LIN {X 0.134,Y -371.526,Z 1771.538,A 0.000,B 0.000,C 90.000,E1 276.777} C_DIS
LIN {X 0.079,Y -367.433,Z 1771.535,A 0.000,B 0.000,C 90.000,E1 276.201} C_DIS
LIN {X 0.001,Y -362.698,Z 1771.531,A 0.000,B 0.000,C 90.000,E1 275.625} C_DIS
LIN {X -0.100,Y -357.339,Z 1771.528,A 0.000,B 0.000,C 90.000,E1 275.049} C_DIS
LIN {X -0.055,Y -351.569,Z 1771.525,A 0.000,B 0.000,C 90.000,E1 274.473} C_DIS
LIN {X -0.094,Y -345.659,Z 1771.522,A 0.000,B 0.000,C 90.000,E1 273.955} C_DIS
LIN {X 0.022,Y -339.520,Z 1771.519,A 0.000,B 0.000,C 90.000,E1 273.440} C_DIS
LIN {X 0.107,Y -330.116,Z 1771.515,A 0.000,B 0.000,C 90.000,E1 272.751} C_DIS
LIN {X 0.126,Y -323.725,Z 1771.513,A 0.000,B 0.000,C 90.000,E1 272.350} C_DIS
LIN {X 0.041,Y -317.098,Z 1771.511,A 0.000,B 0.000,C 90.000,E1 272.007} C_DIS
LIN {X -0.145,Y -310.058,Z 1771.509,A 0.000,B 0.000,C 90.000,E1 271.718} C_DIS
LIN {X -0.066,Y -302.742,Z 1771.508,A 0.000,B 0.000,C 90.000,E1 271.432} C_DIS
LIN {X -0.016,Y -295.334,Z 1771.507,A 0.000,B 0.000,C 90.000,E1 271.203} C_DIS
LIN {X 0.096,Y -283.998,Z 1771.505,A 0.000,B 0.000,C 90.000,E1 270.917} C_DIS
LIN {X -0.066,Y -272.910,Z 1771.504,A 0.000,B 0.000,C 90.000,E1 270.745} C_DIS
LIN {X -0.128,Y -259.523,Z 1771.503,A 0.000,B 0.000,C 90.000,E1 270.573} C_DIS
LIN {X 0.061,Y -245.252,Z 1771.502,A 0.000,B 0.000,C 90.000,E1 270.401} C_DIS
LIN {X 0.075,Y -232.395,Z 1771.502,A 0.000,B 0.000,C 90.000,E1 270.344} C_DIS
LIN {X 0.040,Y -181.579,Z 1771.502,A 0.000,B 0.000,C 90.000,E1 270.344} C_DIS
LIN {X 0.016,Y -180.851,Z 1771.472,A 0.000,B 0.000,C 90.000,E1 264.951} C_DIS
LIN {X 0.098,Y -178.961,Z 1771.444,A 0.000,B 0.000,C 90.000,E1 259.859} C_DIS
LIN {X -0.011,Y -177.369,Z 1771.430,A 0.000,B 0.000,C 90.000,E1 257.353} C_DIS
LIN {X 0.085,Y -175.543,Z 1771.411,A 0.000,B 0.000,C 90.000,E1 253.921} C_DIS
LIN {X -0.076,Y -172.276,Z 1771.387,A 0.000,B 0.000,C 90.000,E1 249.699} C_DIS
LIN {X -0.036,Y -171.755,Z 1771.382,A 0.000,B 0.000,C 90.000,E1 248.827} C_DIS
LIN {X -0.019,Y -167.355,Z 1771.354,A 0.000,B 0.000,C 90.000,E1 243.640} C_DIS
LIN {X 0.063,Y -166.743,Z 1771.349,A 0.000,B 0.000,C 90.000,E1 242.743} C_DIS
LIN {X -0.025,Y -162.722,Z 1771.324,A 0.000,B 0.000,C 90.000,E1 238.408} C_DIS
LIN {X 0.037,Y -161.412,Z 1771.315,A 0.000,B 0.000,C 90.000,E1 236.628} C_DIS
LIN {X 0.078,Y -157.405,Z 1771.290,A 0.000,B 0.000,C 90.000,E1 232.190} C_DIS
LIN {X 0.010,Y -155.405,Z 1771.275,A 0.000,B 0.000,C 90.000,E1 229.542} C_DIS
LIN {X -0.058,Y -151.735,Z 1771.250,A 0.000,B 0.000,C 90.000,E1 225.081} C_DIS
LIN {X -0.046,Y -149.931,Z 1771.235,A 0.000,B 0.000,C 90.000,E1 222.366} C_DIS
LIN {X -0.017,Y -146.781,Z 1771.210,A 0.000,B 0.000,C 90.000,E1 217.810} C_DIS
LIN {X 0.086,Y -145.353,Z 1771.195,A 0.000,B 0.000,C 90.000,E1 215.025} C_DIS
LIN {X 0.001,Y -142.425,Z 1771.164,A 0.000,B 0.000,C 90.000,E1 209.539} C_DIS
LIN {X 0.050,Y -141.412,Z 1771.149,A 0.000,B 0.000,C 90.000,E1 206.744} C_DIS
LIN {X 0.037,Y -139.359,Z 1771.113,A 0.000,B 0.000,C 90.000,E1 200.248} C_DIS
LIN {X 0.025,Y -138.802,Z 1771.097,A 0.000,B 0.000,C 90.000,E1 197.457} C_DIS
LIN {X -0.056,Y -138.349,Z 1771.056,A 0.000,B 0.000,C 90.000,E1 190.018} C_DIS
LIN {X -0.042,Y -139.366,Z 1771.009,A 0.000,B 0.000,C 90.000,E1 181.604} C_DIS
LIN {X 0.011,Y -141.254,Z 1770.973,A 0.000,B 0.000,C 90.000,E1 175.065} C_DIS
LIN {X -0.030,Y -142.621,Z 1770.957,A 0.000,B 0.000,C 90.000,E1 172.299} C_DIS
LIN {X 0.063,Y -144.941,Z 1770.932,A 0.000,B 0.000,C 90.000,E1 167.645} C_DIS
LIN {X 0.055,Y -147.571,Z 1770.911,A 0.000,B 0.000,C 90.000,E1 163.976} C_DIS
LIN {X -0.055,Y -150.179,Z 1770.891,A 0.000,B 0.000,C 90.000,E1 160.369} C_DIS
LIN {X -0.048,Y -153.556,Z 1770.871,A 0.000,B 0.000,C 90.000,E1 156.741} C_DIS
LIN {X 0.004,Y -156.974,Z 1770.851,A 0.000,B 0.000,C 90.000,E1 153.127} C_DIS
LIN {X 0.078,Y -161.085,Z 1770.831,A 0.000,B 0.000,C 90.000,E1 149.537} C_DIS
LIN {X 0.023,Y -163.189,Z 1770.821,A 0.000,B 0.000,C 90.000,E1 147.788} C_DIS
LIN {X 0.029,Y -167.613,Z 1770.802,A 0.000,B 0.000,C 90.000,E1 144.276} C_DIS
LIN {X -0.061,Y -171.441,Z 1770.787,A 0.000,B 0.000,C 90.000,E1 141.698} C_DIS
LIN {X -0.024,Y -176.363,Z 1770.768,A 0.000,B 0.000,C 90.000,E1 138.243} C_DIS
LIN {X 0.098,Y -180.654,Z 1770.754,A 0.000,B 0.000,C 90.000,E1 135.648} C_DIS
LIN {X 0.082,Y -186.056,Z 1770.735,A 0.000,B 0.000,C 90.000,E1 132.285} C_DIS
LIN {X 0.019,Y -190.693,Z 1770.721,A 0.000,B 0.000,C 90.000,E1 129.806} C_DIS
LIN {X 0.051,Y -196.444,Z 1770.703,A 0.000,B 0.000,C 90.000,E1 126.503} C_DIS
LIN {X 0.018,Y -201.228,Z 1770.689,A 0.000,B 0.000,C 90.000,E1 124.072} C_DIS
LIN {X -0.054,Y -207.184,Z 1770.671,A 0.000,B 0.000,C 90.000,E1 120.875} C_DIS
LIN {X 0.039,Y -210.847,Z 1770.661,A 0.000,B 0.000,C 90.000,E1 119.027} C_DIS
LIN {X 0.028,Y -337.420,Z 1770.661,A 0.000,B 0.000,C 90.000,E1 119.027} C_DIS
LIN {X -0.089,Y -339.869,Z 1770.661,A 0.000,B 0.000,C 90.000,E1 118.999} C_DIS
LIN {X -0.080,Y -344.748,Z 1770.660,A 0.000,B 0.000,C 90.000,E1 118.743} C_DIS
LIN {X -0.070,Y -347.508,Z 1770.658,A 0.000,B 0.000,C 90.000,E1 118.487} C_DIS
LIN {X -0.087,Y -351.162,Z 1770.655,A 0.000,B 0.000,C 90.000,E1 117.975} C_DIS
LIN {X 0.074,Y -367.528,Z 1770.637,A 0.000,B 0.000,C 90.000,E1 114.643} C_DIS
LIN {X -0.051,Y -382.548,Z 1770.622,A 0.000,B 0.000,C 90.000,E1 112.025} C_DIS
LIN {X -0.218,Y -397.315,Z 1770.610,A 0.000,B 0.000,C 90.000,E1 109.758} C_DIS
LIN {X -0.163,Y -413.522,Z 1770.597,A 0.000,B 0.000,C 90.000,E1 107.511} C_DIS
LIN {X 0.213,Y -432.981,Z 1770.583,A 0.000,B 0.000,C 90.000,E1 105.009} C_DIS
LIN {X -0.177,Y -450.867,Z 1770.572,A 0.000,B 0.000,C 90.000,E1 102.939} C_DIS
LIN {X -0.211,Y -466.762,Z 1770.562,A 0.000,B 0.000,C 90.000,E1 101.130} C_DIS
LIN {X 0.223,Y -480.264,Z 1770.553,A 0.000,B 0.000,C 90.000,E1 99.557} C_DIS
LIN {X 0.145,Y -488.951,Z 1770.548,A 0.000,B 0.000,C 90.000,E1 98.568} C_DIS
LIN {X 0.255,Y -495.091,Z 1770.544,A 0.000,B 0.000,C 90.000,E1 97.814} C_DIS
LIN {X -0.146,Y -500.631,Z 1770.540,A 0.000,B 0.000,C 90.000,E1 97.125} C_DIS
LIN {X 0.135,Y -503.706,Z 1770.537,A 0.000,B 0.000,C 90.000,E1 96.606} C_DIS
LIN {X -0.065,Y -505.070,Z 1770.534,A 0.000,B 0.000,C 90.000,E1 96.144} C_DIS
LIN {X 0.244,Y -503.625,Z 1770.531,A 0.000,B 0.000,C 90.000,E1 95.625} C_DIS
LIN {X 0.057,Y -501.685,Z 1770.529,A 0.000,B 0.000,C 90.000,E1 95.163} C_DIS
LIN {X 0.114,Y -497.247,Z 1770.523,A 0.000,B 0.000,C 90.000,E1 94.188} C_DIS
LIN {X 0.113,Y -492.374,Z 1770.518,A 0.000,B 0.000,C 90.000,E1 93.212} C_DIS
LIN {X 0.059,Y -487.076,Z 1770.512,A 0.000,B 0.000,C 90.000,E1 92.236} C_DIS
LIN {X 0.091,Y -478.578,Z 1770.504,A 0.000,B 0.000,C 90.000,E1 90.745} C_DIS
LIN {X -0.031,Y -469.762,Z 1770.496,A 0.000,B 0.000,C 90.000,E1 89.255} C_DIS
LIN {X 0.173,Y -460.513,Z 1770.487,A 0.000,B 0.000,C 90.000,E1 87.707} C_DIS
LIN {X 0.211,Y -451.010,Z 1770.479,A 0.000,B 0.000,C 90.000,E1 86.159} C_DIS
LIN {X 0.107,Y -441.181,Z 1770.470,A 0.000,B 0.000,C 90.000,E1 84.609} C_DIS
LIN {X 0.063,Y -429.518,Z 1770.460,A 0.000,B 0.000,C 90.000,E1 82.761} C_DIS
LIN {X -0.141,Y -417.733,Z 1770.449,A 0.000,B 0.000,C 90.000,E1 80.905} C_DIS
LIN {X -0.067,Y -404.294,Z 1770.437,A 0.000,B 0.000,C 90.000,E1 78.701} C_DIS
LIN {X 0.042,Y -388.295,Z 1770.422,A 0.000,B 0.000,C 90.000,E1 75.880} C_DIS
LIN {X -0.027,Y -371.685,Z 1770.404,A 0.000,B 0.000,C 90.000,E1 72.725} C_DIS
LIN {X -0.022,Y -360.102,Z 1770.391,A 0.000,B 0.000,C 90.000,E1 70.369} C_DIS
LIN {X -0.051,Y -348.781,Z 1770.378,A 0.000,B 0.000,C 90.000,E1 67.975} C_DIS
LIN {X -0.084,Y -336.469,Z 1770.362,A 0.000,B 0.000,C 90.000,E1 65.229} C_DIS
LIN {X -0.132,Y -325.824,Z 1770.348,A 0.000,B 0.000,C 90.000,E1 62.743} C_DIS
LIN {X 0.044,Y -319.126,Z 1770.340,A 0.000,B 0.000,C 90.000,E1 61.129} C_DIS
LIN {X 0.054,Y -310.757,Z 1770.329,A 0.000,B 0.000,C 90.000,E1 59.203} C_DIS
LIN {X 0.070,Y -301.966,Z 1770.318,A 0.000,B 0.000,C 90.000,E1 57.248} C_DIS
LIN {X 0.000,Y -290.001,Z 1770.303,A 0.000,B 0.000,C 90.000,E1 54.609} C_DIS
LIN {X -0.025,Y -278.506,Z 1770.288,A 0.000,B 0.000,C 90.000,E1 51.904} C_DIS
LIN {X 0.046,Y -266.203,Z 1770.271,A 0.000,B 0.000,C 90.000,E1 48.771} C_DIS
LIN {X -0.111,Y -255.809,Z 1770.255,A 0.000,B 0.000,C 90.000,E1 45.972} C_DIS
LIN {X 0.004,Y -244.440,Z 1770.237,A 0.000,B 0.000,C 90.000,E1 42.690} C_DIS
LIN {X 0.040,Y -234.846,Z 1770.221,A 0.000,B 0.000,C 90.000,E1 39.725} C_DIS
LIN {X -0.011,Y -224.683,Z 1770.202,A 0.000,B 0.000,C 90.000,E1 36.343} C_DIS
LIN {X -0.086,Y -216.282,Z 1770.185,A 0.000,B 0.000,C 90.000,E1 33.293} C_DIS
LIN {X 0.061,Y -208.453,Z 1770.167,A 0.000,B 0.000,C 90.000,E1 30.129} C_DIS
LIN {X 0.065,Y -201.341,Z 1770.150,A 0.000,B 0.000,C 90.000,E1 26.950} C_DIS
LIN {X -0.098,Y -194.992,Z 1770.132,A 0.000,B 0.000,C 90.000,E1 23.770} C_DIS
LIN {X -0.038,Y -189.466,Z 1770.114,A 0.000,B 0.000,C 90.000,E1 20.482} C_DIS
LIN {X -0.021,Y -184.796,Z 1770.095,A 0.000,B 0.000,C 90.000,E1 17.166} C_DIS
LIN {X -0.044,Y -181.068,Z 1770.077,A 0.000,B 0.000,C 90.000,E1 13.828} C_DIS
LIN {X -0.060,Y -177.501,Z 1770.053,A 0.000,B 0.000,C 90.000,E1 9.613} C_DIS
LIN {X 0.038,Y -174.559,Z 1770.025,A 0.000,B 0.000,C 90.000,E1 4.473} C_DIS
LIN {X -0.019,Y -172.925,Z 1769.983,A 0.000,B 0.000,C 90.000,E1 356.963} C_DIS
LIN {X -0.075,Y -173.224,Z 1769.950,A 0.000,B 0.000,C 90.000,E1 350.971} C_DIS
LIN {X -0.040,Y -175.130,Z 1769.912,A 0.000,B 0.000,C 90.000,E1 344.102} C_DIS
LIN {X 0.050,Y -178.027,Z 1769.883,A 0.000,B 0.000,C 90.000,E1 338.954} C_DIS
LIN {X -0.020,Y -181.888,Z 1769.855,A 0.000,B 0.000,C 90.000,E1 333.896} C_DIS
LIN {X 0.087,Y -186.053,Z 1769.832,A 0.000,B 0.000,C 90.000,E1 329.665} C_DIS
LIN {X -0.032,Y -190.201,Z 1769.813,A 0.000,B 0.000,C 90.000,E1 326.373} C_DIS
LIN {X 0.058,Y -195.220,Z 1769.795,A 0.000,B 0.000,C 90.000,E1 323.050} C_DIS
LIN {X -0.081,Y -199.651,Z 1769.781,A 0.000,B 0.000,C 90.000,E1 320.642} C_DIS
LIN {X 0.117,Y -204.814,Z 1769.768,A 0.000,B 0.000,C 90.000,E1 318.162} C_DIS
LIN {X -0.011,Y -211.724,Z 1769.752,A 0.000,B 0.000,C 90.000,E1 315.405} C_DIS
LIN {X -0.093,Y -217.337,Z 1769.741,A 0.000,B 0.000,C 90.000,E1 313.461} C_DIS
LIN {X -0.077,Y -223.801,Z 1769.730,A 0.000,B 0.000,C 90.000,E1 311.515} C_DIS
LIN {X -0.026,Y -229.683,Z 1769.722,A 0.000,B 0.000,C 90.000,E1 309.967} C_DIS
LIN {X -0.075,Y -236.287,Z 1769.714,A 0.000,B 0.000,C 90.000,E1 308.463} C_DIS
LIN {X -0.003,Y -243.650,Z 1769.705,A 0.000,B 0.000,C 90.000,E1 306.950} C_DIS
LIN {X 0.026,Y -253.717,Z 1769.695,A 0.000,B 0.000,C 90.000,E1 305.105} C_DIS
LIN {X -0.064,Y -271.589,Z 1769.679,A 0.000,B 0.000,C 90.000,E1 302.260} C_DIS
LIN {X 0.107,Y -291.086,Z 1769.664,A 0.000,B 0.000,C 90.000,E1 299.461} C_DIS
LIN {X 0.090,Y -309.111,Z 1769.651,A 0.000,B 0.000,C 90.000,E1 297.129} C_DIS
LIN {X 0.060,Y -324.890,Z 1769.640,A 0.000,B 0.000,C 90.000,E1 295.207} C_DIS
LIN {X -0.029,Y -338.121,Z 1769.631,A 0.000,B 0.000,C 90.000,E1 293.643} C_DIS
LIN {X 0.097,Y -350.912,Z 1769.623,A 0.000,B 0.000,C 90.000,E1 292.078} C_DIS
LIN {X -0.181,Y -363.260,Z 1769.614,A 0.000,B 0.000,C 90.000,E1 290.610} C_DIS
LIN {X 0.028,Y -370.117,Z 1769.609,A 0.000,B 0.000,C 90.000,E1 289.685} C_DIS
LIN {X 0.175,Y -376.215,Z 1769.604,A 0.000,B 0.000,C 90.000,E1 288.779} C_DIS
LIN {X -0.088,Y -381.405,Z 1769.600,A 0.000,B 0.000,C 90.000,E1 287.946} C_DIS
LIN {X 0.174,Y -385.621,Z 1769.595,A 0.000,B 0.000,C 90.000,E1 287.040} C_DIS
LIN {X -0.035,Y -387.867,Z 1769.592,A 0.000,B 0.000,C 90.000,E1 286.496} C_DIS
LIN {X 0.142,Y -389.790,Z 1769.588,A 0.000,B 0.000,C 90.000,E1 285.898} C_DIS
LIN {X -0.156,Y -391.399,Z 1769.585,A 0.000,B 0.000,C 90.000,E1 285.371} C_DIS
LIN {X 0.039,Y -392.646,Z 1769.582,A 0.000,B 0.000,C 90.000,E1 284.773} C_DIS
LIN {X 0.146,Y -393.497,Z 1769.579,A 0.000,B 0.000,C 90.000,E1 284.189} C_DIS
LIN {X -0.026,Y -394.043,Z 1769.576,A 0.000,B 0.000,C 90.000,E1 283.647} C_DIS
LIN {X 0.096,Y -394.159,Z 1769.573,A 0.000,B 0.000,C 90.000,E1 283.063} C_DIS
LIN {X -0.161,Y -393.968,Z 1769.569,A 0.000,B 0.000,C 90.000,E1 282.535} C_DIS
LIN {X -0.032,Y -393.368,Z 1769.566,A 0.000,B 0.000,C 90.000,E1 281.951} C_DIS
LIN {X 0.097,Y -392.395,Z 1769.563,A 0.000,B 0.000,C 90.000,E1 281.366} C_DIS
LIN {X -0.164,Y -391.035,Z 1769.560,A 0.000,B 0.000,C 90.000,E1 280.838} C_DIS
LIN {X -0.046,Y -389.272,Z 1769.557,A 0.000,B 0.000,C 90.000,E1 280.254} C_DIS
LIN {X 0.104,Y -385.801,Z 1769.552,A 0.000,B 0.000,C 90.000,E1 279.378} C_DIS
LIN {X 0.158,Y -381.625,Z 1769.547,A 0.000,B 0.000,C 90.000,E1 278.511} C_DIS
LIN {X 0.173,Y -376.958,Z 1769.543,A 0.000,B 0.000,C 90.000,E1 277.644} C_DIS
LIN {X 0.151,Y -371.653,Z 1769.538,A 0.000,B 0.000,C 90.000,E1 276.777} C_DIS
LIN {X 0.096,Y -367.561,Z 1769.535,A 0.000,B 0.000,C 90.000,E1 276.201} C_DIS
LIN {X 0.019,Y -362.844,Z 1769.531,A 0.000,B 0.000,C 90.000,E1 275.625} C_DIS
LIN {X -0.081,Y -357.478,Z 1769.528,A 0.000,B 0.000,C 90.000,E1 275.049} C_DIS
LIN {X -0.037,Y -351.680,Z 1769.525,A 0.000,B 0.000,C 90.000,E1 274.473} C_DIS
LIN {X -0.052,Y -345.790,Z 1769.522,A 0.000,B 0.000,C 90.000,E1 273.955} C_DIS
LIN {X 0.084,Y -339.650,Z 1769.519,A 0.000,B 0.000,C 90.000,E1 273.440} C_DIS
LIN {X -0.134,Y -330.302,Z 1769.516,A 0.000,B 0.000,C 90.000,E1 272.808} C_DIS
LIN {X -0.135,Y -323.834,Z 1769.513,A 0.000,B 0.000,C 90.000,E1 272.407} C_DIS
LIN {X 0.090,Y -317.201,Z 1769.511,A 0.000,B 0.000,C 90.000,E1 272.007} C_DIS
LIN {X -0.087,Y -310.184,Z 1769.509,A 0.000,B 0.000,C 90.000,E1 271.718} C_DIS
LIN {X 0.014,Y -303.034,Z 1769.508,A 0.000,B 0.000,C 90.000,E1 271.432} C_DIS
LIN {X 0.065,Y -295.721,Z 1769.507,A 0.000,B 0.000,C 90.000,E1 271.203} C_DIS
LIN {X -0.114,Y -284.435,Z 1769.505,A 0.000,B 0.000,C 90.000,E1 270.974} C_DIS
LIN {X -0.027,Y -272.894,Z 1769.504,A 0.000,B 0.000,C 90.000,E1 270.745} C_DIS
LIN {X -0.086,Y -259.438,Z 1769.503,A 0.000,B 0.000,C 90.000,E1 270.573} C_DIS
LIN {X 0.099,Y -244.528,Z 1769.502,A 0.000,B 0.000,C 90.000,E1 270.401} C_DIS
LIN {X -0.093,Y -233.131,Z 1769.502,A 0.000,B 0.000,C 90.000,E1 270.401} C_DIS
LIN {X 0.073,Y -181.578,Z 1769.502,A 0.000,B 0.000,C 90.000,E1 270.344} C_DIS
LIN {X 0.050,Y -180.854,Z 1769.472,A 0.000,B 0.000,C 90.000,E1 264.951} C_DIS
LIN {X -0.076,Y -178.965,Z 1769.444,A 0.000,B 0.000,C 90.000,E1 259.926} C_DIS
LIN {X -0.066,Y -177.916,Z 1769.434,A 0.000,B 0.000,C 90.000,E1 258.229} C_DIS
LIN {X -0.050,Y -175.552,Z 1769.411,A 0.000,B 0.000,C 90.000,E1 253.976} C_DIS
LIN {X -0.043,Y -172.283,Z 1769.387,A 0.000,B 0.000,C 90.000,E1 249.699} C_DIS
LIN {X -0.002,Y -171.762,Z 1769.382,A 0.000,B 0.000,C 90.000,E1 248.827} C_DIS
LIN {X 0.014,Y -167.362,Z 1769.354,A 0.000,B 0.000,C 90.000,E1 243.640} C_DIS
LIN {X -0.053,Y -166.751,Z 1769.349,A 0.000,B 0.000,C 90.000,E1 242.794} C_DIS
LIN {X 0.007,Y -162.730,Z 1769.324,A 0.000,B 0.000,C 90.000,E1 238.408} C_DIS
LIN {X 0.068,Y -161.421,Z 1769.315,A 0.000,B 0.000,C 90.000,E1 236.628} C_DIS
LIN {X -0.015,Y -157.415,Z 1769.290,A 0.000,B 0.000,C 90.000,E1 232.236} C_DIS
LIN {X 0.042,Y -155.416,Z 1769.275,A 0.000,B 0.000,C 90.000,E1 229.542} C_DIS
LIN {X -0.027,Y -151.743,Z 1769.250,A 0.000,B 0.000,C 90.000,E1 225.081} C_DIS
LIN {X -0.015,Y -149.941,Z 1769.235,A 0.000,B 0.000,C 90.000,E1 222.366} C_DIS
LIN {X 0.013,Y -146.788,Z 1769.210,A 0.000,B 0.000,C 90.000,E1 217.810} C_DIS
LIN {X -0.087,Y -145.361,Z 1769.195,A 0.000,B 0.000,C 90.000,E1 215.105} C_DIS
LIN {X 0.030,Y -142.430,Z 1769.164,A 0.000,B 0.000,C 90.000,E1 209.539} C_DIS
LIN {X -0.047,Y -141.418,Z 1769.149,A 0.000,B 0.000,C 90.000,E1 206.796} C_DIS
LIN {X -0.064,Y -139.361,Z 1769.113,A 0.000,B 0.000,C 90.000,E1 200.301} C_DIS
LIN {X 0.054,Y -138.804,Z 1769.097,A 0.000,B 0.000,C 90.000,E1 197.457} C_DIS
LIN {X -0.027,Y -138.350,Z 1769.056,A 0.000,B 0.000,C 90.000,E1 190.018} C_DIS
LIN {X -0.052,Y -139.545,Z 1769.004,A 0.000,B 0.000,C 90.000,E1 180.688} C_DIS
LIN {X 0.041,Y -141.248,Z 1768.973,A 0.000,B 0.000,C 90.000,E1 175.065} C_DIS
LIN {X -0.001,Y -142.617,Z 1768.957,A 0.000,B 0.000,C 90.000,E1 172.299} C_DIS
LIN {X -0.049,Y -144.934,Z 1768.932,A 0.000,B 0.000,C 90.000,E1 167.701} C_DIS
LIN {X -0.056,Y -147.563,Z 1768.911,A 0.000,B 0.000,C 90.000,E1 164.031} C_DIS
LIN {X -0.025,Y -150.170,Z 1768.891,A 0.000,B 0.000,C 90.000,E1 160.369} C_DIS
LIN {X -0.016,Y -153.545,Z 1768.871,A 0.000,B 0.000,C 90.000,E1 156.741} C_DIS
LIN {X 0.036,Y -156.962,Z 1768.851,A 0.000,B 0.000,C 90.000,E1 153.127} C_DIS
LIN {X -0.029,Y -161.070,Z 1768.831,A 0.000,B 0.000,C 90.000,E1 149.587} C_DIS
LIN {X 0.056,Y -163.177,Z 1768.821,A 0.000,B 0.000,C 90.000,E1 147.788} C_DIS
LIN {X 0.062,Y -167.597,Z 1768.802,A 0.000,B 0.000,C 90.000,E1 144.276} C_DIS
LIN {X -0.028,Y -171.426,Z 1768.787,A 0.000,B 0.000,C 90.000,E1 141.698} C_DIS
LIN {X 0.010,Y -176.345,Z 1768.768,A 0.000,B 0.000,C 90.000,E1 138.243} C_DIS
LIN {X 0.006,Y -180.635,Z 1768.754,A 0.000,B 0.000,C 90.000,E1 135.688} C_DIS
LIN {X -0.009,Y -186.037,Z 1768.735,A 0.000,B 0.000,C 90.000,E1 132.324} C_DIS
LIN {X 0.055,Y -190.673,Z 1768.721,A 0.000,B 0.000,C 90.000,E1 129.806} C_DIS
LIN {X 0.088,Y -196.424,Z 1768.703,A 0.000,B 0.000,C 90.000,E1 126.503} C_DIS
LIN {X 0.054,Y -201.211,Z 1768.689,A 0.000,B 0.000,C 90.000,E1 124.072} C_DIS
LIN {X -0.017,Y -207.163,Z 1768.672,A 0.000,B 0.000,C 90.000,E1 120.875} C_DIS
LIN {X -0.048,Y -210.802,Z 1768.661,A 0.000,B 0.000,C 90.000,E1 119.077} C_DIS
LIN {X -0.125,Y -337.161,Z 1768.661,A 0.000,B 0.000,C 90.000,E1 119.077} C_DIS
LIN {X 0.051,Y -342.194,Z 1768.661,A 0.000,B 0.000,C 90.000,E1 118.899} C_DIS
LIN {X 0.142,Y -344.436,Z 1768.660,A 0.000,B 0.000,C 90.000,E1 118.743} C_DIS
LIN {X -0.008,Y -347.499,Z 1768.658,A 0.000,B 0.000,C 90.000,E1 118.487} C_DIS
LIN {X -0.016,Y -351.099,Z 1768.655,A 0.000,B 0.000,C 90.000,E1 117.975} C_DIS
LIN {X 0.145,Y -367.446,Z 1768.637,A 0.000,B 0.000,C 90.000,E1 114.643} C_DIS
LIN {X 0.021,Y -382.458,Z 1768.622,A 0.000,B 0.000,C 90.000,E1 112.025} C_DIS
LIN {X -0.145,Y -397.219,Z 1768.610,A 0.000,B 0.000,C 90.000,E1 109.758} C_DIS
LIN {X -0.090,Y -413.419,Z 1768.597,A 0.000,B 0.000,C 90.000,E1 107.511} C_DIS
LIN {X 0.047,Y -435.616,Z 1768.582,A 0.000,B 0.000,C 90.000,E1 104.773} C_DIS
LIN {X 0.155,Y -454.157,Z 1768.570,A 0.000,B 0.000,C 90.000,E1 102.647} C_DIS
LIN {X 0.214,Y -470.696,Z 1768.560,A 0.000,B 0.000,C 90.000,E1 100.838} C_DIS
LIN {X 0.256,Y -484.880,Z 1768.552,A 0.000,B 0.000,C 90.000,E1 99.321} C_DIS
LIN {X 0.058,Y -496.414,Z 1768.545,A 0.000,B 0.000,C 90.000,E1 98.106} C_DIS
LIN {X 0.091,Y -505.123,Z 1768.540,A 0.000,B 0.000,C 90.000,E1 97.125} C_DIS
LIN {X 0.024,Y -507.149,Z 1768.538,A 0.000,B 0.000,C 90.000,E1 96.891} C_DIS
LIN {X -0.105,Y -508.531,Z 1768.537,A 0.000,B 0.000,C 90.000,E1 96.663} C_DIS
LIN {X 0.226,Y -509.449,Z 1768.534,A 0.000,B 0.000,C 90.000,E1 96.144} C_DIS
LIN {X 0.059,Y -508.348,Z 1768.532,A 0.000,B 0.000,C 90.000,E1 95.682} C_DIS
LIN {X 0.104,Y -501.995,Z 1768.525,A 0.000,B 0.000,C 90.000,E1 94.473} C_DIS
LIN {X -0.077,Y -493.931,Z 1768.517,A 0.000,B 0.000,C 90.000,E1 93.037} C_DIS
LIN {X 0.221,Y -486.722,Z 1768.510,A 0.000,B 0.000,C 90.000,E1 91.776} C_DIS
LIN {X 0.054,Y -476.160,Z 1768.500,A 0.000,B 0.000,C 90.000,E1 90.057} C_DIS
LIN {X -0.110,Y -466.812,Z 1768.492,A 0.000,B 0.000,C 90.000,E1 88.568} C_DIS
LIN {X 0.039,Y -457.124,Z 1768.484,A 0.000,B 0.000,C 90.000,E1 87.020} C_DIS
LIN {X 0.044,Y -447.200,Z 1768.475,A 0.000,B 0.000,C 90.000,E1 85.469} C_DIS
LIN {X 0.080,Y -435.274,Z 1768.465,A 0.000,B 0.000,C 90.000,E1 83.628} C_DIS
LIN {X -0.187,Y -424.927,Z 1768.456,A 0.000,B 0.000,C 90.000,E1 82.064} C_DIS
LIN {X 0.065,Y -411.129,Z 1768.444,A 0.000,B 0.000,C 90.000,E1 79.859} C_DIS
LIN {X -0.107,Y -393.082,Z 1768.427,A 0.000,B 0.000,C 90.000,E1 76.825} C_DIS
LIN {X -0.116,Y -376.155,Z 1768.409,A 0.000,B 0.000,C 90.000,E1 73.685} C_DIS
LIN {X -0.002,Y -364.410,Z 1768.396,A 0.000,B 0.000,C 90.000,E1 71.329} C_DIS
LIN {X -0.001,Y -351.560,Z 1768.381,A 0.000,B 0.000,C 90.000,E1 68.646} C_DIS
LIN {X -0.092,Y -337.738,Z 1768.364,A 0.000,B 0.000,C 90.000,E1 65.613} C_DIS
LIN {X -0.111,Y -327.062,Z 1768.351,A 0.000,B 0.000,C 90.000,E1 63.127} C_DIS
LIN {X 0.177,Y -319.049,Z 1768.340,A 0.000,B 0.000,C 90.000,E1 61.179} C_DIS
LIN {X 0.028,Y -310.746,Z 1768.329,A 0.000,B 0.000,C 90.000,E1 59.282} C_DIS
LIN {X 0.040,Y -301.935,Z 1768.318,A 0.000,B 0.000,C 90.000,E1 57.327} C_DIS
LIN {X -0.033,Y -290.000,Z 1768.304,A 0.000,B 0.000,C 90.000,E1 54.689} C_DIS
LIN {X -0.059,Y -278.512,Z 1768.289,A 0.000,B 0.000,C 90.000,E1 51.984} C_DIS
LIN {X -0.068,Y -267.546,Z 1768.273,A 0.000,B 0.000,C 90.000,E1 49.218} C_DIS
LIN {X 0.003,Y -257.069,Z 1768.258,A 0.000,B 0.000,C 90.000,E1 46.377} C_DIS
LIN {X -0.029,Y -245.621,Z 1768.240,A 0.000,B 0.000,C 90.000,E1 43.137} C_DIS
LIN {X 0.033,Y -235.942,Z 1768.223,A 0.000,B 0.000,C 90.000,E1 40.172} C_DIS
LIN {X 0.066,Y -226.735,Z 1768.207,A 0.000,B 0.000,C 90.000,E1 37.156} C_DIS
LIN {X -0.019,Y -218.172,Z 1768.190,A 0.000,B 0.000,C 90.000,E1 34.119} C_DIS
LIN {X -0.005,Y -210.200,Z 1768.172,A 0.000,B 0.000,C 90.000,E1 31.003} C_DIS
LIN {X -0.036,Y -202.870,Z 1768.155,A 0.000,B 0.000,C 90.000,E1 27.847} C_DIS
LIN {X -0.076,Y -196.370,Z 1768.137,A 0.000,B 0.000,C 90.000,E1 24.643} C_DIS
LIN {X 0.016,Y -190.612,Z 1768.119,A 0.000,B 0.000,C 90.000,E1 21.354} C_DIS
LIN {X 0.007,Y -185.697,Z 1768.100,A 0.000,B 0.000,C 90.000,E1 18.055} C_DIS
LIN {X 0.001,Y -181.730,Z 1768.082,A 0.000,B 0.000,C 90.000,E1 14.717} C_DIS
LIN {X 0.043,Y -177.905,Z 1768.058,A 0.000,B 0.000,C 90.000,E1 10.489} C_DIS
LIN {X -0.014,Y -175.134,Z 1768.035,A 0.000,B 0.000,C 90.000,E1 6.258} C_DIS
LIN {X -0.031,Y -172.984,Z 1767.997,A 0.000,B 0.000,C 90.000,E1 359.542} C_DIS
LIN {X 0.035,Y -172.749,Z 1767.959,A 0.000,B 0.000,C 90.000,E1 352.648} C_DIS
LIN {X -0.057,Y -174.214,Z 1767.921,A 0.000,B 0.000,C 90.000,E1 345.811} C_DIS
LIN {X -0.047,Y -176.679,Z 1767.893,A 0.000,B 0.000,C 90.000,E1 340.678} C_DIS
LIN {X 0.087,Y -180.274,Z 1767.864,A 0.000,B 0.000,C 90.000,E1 335.537} C_DIS
LIN {X -0.108,Y -184.088,Z 1767.841,A 0.000,B 0.000,C 90.000,E1 331.385} C_DIS
LIN {X 0.024,Y -188.975,Z 1767.818,A 0.000,B 0.000,C 90.000,E1 327.168} C_DIS
LIN {X 0.022,Y -193.826,Z 1767.799,A 0.000,B 0.000,C 90.000,E1 323.863} C_DIS
LIN {X 0.009,Y -199.668,Z 1767.781,A 0.000,B 0.000,C 90.000,E1 320.598} C_DIS
LIN {X 0.051,Y -204.876,Z 1767.768,A 0.000,B 0.000,C 90.000,E1 318.162} C_DIS
LIN {X -0.078,Y -211.820,Z 1767.752,A 0.000,B 0.000,C 90.000,E1 315.405} C_DIS
LIN {X -0.001,Y -217.484,Z 1767.741,A 0.000,B 0.000,C 90.000,E1 313.419} C_DIS
LIN {X 0.024,Y -223.986,Z 1767.730,A 0.000,B 0.000,C 90.000,E1 311.472} C_DIS
LIN {X 0.056,Y -229.894,Z 1767.722,A 0.000,B 0.000,C 90.000,E1 309.930} C_DIS
LIN {X -0.140,Y -236.530,Z 1767.714,A 0.000,B 0.000,C 90.000,E1 308.463} C_DIS
LIN {X -0.086,Y -245.869,Z 1767.703,A 0.000,B 0.000,C 90.000,E1 306.583} C_DIS
LIN {X -0.149,Y -258.327,Z 1767.691,A 0.000,B 0.000,C 90.000,E1 304.405} C_DIS
LIN {X -0.044,Y -276.646,Z 1767.675,A 0.000,B 0.000,C 90.000,E1 301.544} C_DIS
LIN {X -0.128,Y -296.568,Z 1767.660,A 0.000,B 0.000,C 90.000,E1 298.821} C_DIS
LIN {X -0.032,Y -314.755,Z 1767.647,A 0.000,B 0.000,C 90.000,E1 296.488} C_DIS
LIN {X -0.047,Y -327.918,Z 1767.638,A 0.000,B 0.000,C 90.000,E1 294.899} C_DIS
LIN {X -0.065,Y -341.055,Z 1767.630,A 0.000,B 0.000,C 90.000,E1 293.334} C_DIS
LIN {X 0.116,Y -353.763,Z 1767.621,A 0.000,B 0.000,C 90.000,E1 291.770} C_DIS
LIN {X -0.176,Y -363.608,Z 1767.614,A 0.000,B 0.000,C 90.000,E1 290.610} C_DIS
LIN {X 0.037,Y -370.447,Z 1767.609,A 0.000,B 0.000,C 90.000,E1 289.685} C_DIS
LIN {X 0.187,Y -376.555,Z 1767.604,A 0.000,B 0.000,C 90.000,E1 288.779} C_DIS
LIN {X -0.075,Y -380.120,Z 1767.601,A 0.000,B 0.000,C 90.000,E1 288.236} C_DIS
LIN {X 0.062,Y -384.652,Z 1767.596,A 0.000,B 0.000,C 90.000,E1 287.347} C_DIS
LIN {X -0.152,Y -387.147,Z 1767.593,A 0.000,B 0.000,C 90.000,E1 286.804} C_DIS
LIN {X 0.164,Y -390.154,Z 1767.589,A 0.000,B 0.000,C 90.000,E1 285.898} C_DIS
LIN {X -0.132,Y -391.737,Z 1767.585,A 0.000,B 0.000,C 90.000,E1 285.371} C_DIS
LIN {X 0.066,Y -392.961,Z 1767.582,A 0.000,B 0.000,C 90.000,E1 284.773} C_DIS
LIN {X -0.207,Y -393.853,Z 1767.579,A 0.000,B 0.000,C 90.000,E1 284.245} C_DIS
LIN {X 0.005,Y -394.374,Z 1767.576,A 0.000,B 0.000,C 90.000,E1 283.647} C_DIS
LIN {X 0.129,Y -394.501,Z 1767.573,A 0.000,B 0.000,C 90.000,E1 283.063} C_DIS
LIN {X -0.126,Y -394.317,Z 1767.570,A 0.000,B 0.000,C 90.000,E1 282.535} C_DIS
LIN {X 0.005,Y -393.704,Z 1767.566,A 0.000,B 0.000,C 90.000,E1 281.951} C_DIS
LIN {X 0.135,Y -392.724,Z 1767.563,A 0.000,B 0.000,C 90.000,E1 281.366} C_DIS
LIN {X -0.123,Y -391.333,Z 1767.560,A 0.000,B 0.000,C 90.000,E1 280.838} C_DIS
LIN {X -0.003,Y -389.523,Z 1767.557,A 0.000,B 0.000,C 90.000,E1 280.254} C_DIS
LIN {X 0.149,Y -385.978,Z 1767.552,A 0.000,B 0.000,C 90.000,E1 279.378} C_DIS
LIN {X -0.146,Y -380.185,Z 1767.546,A 0.000,B 0.000,C 90.000,E1 278.276} C_DIS
LIN {X -0.137,Y -375.367,Z 1767.541,A 0.000,B 0.000,C 90.000,E1 277.409} C_DIS
LIN {X 0.191,Y -369.834,Z 1767.536,A 0.000,B 0.000,C 90.000,E1 276.486} C_DIS
LIN {X 0.122,Y -365.432,Z 1767.533,A 0.000,B 0.000,C 90.000,E1 275.910} C_DIS
LIN {X 0.032,Y -360.468,Z 1767.530,A 0.000,B 0.000,C 90.000,E1 275.334} C_DIS
LIN {X 0.018,Y -354.903,Z 1767.526,A 0.000,B 0.000,C 90.000,E1 274.759} C_DIS
LIN {X -0.160,Y -349.006,Z 1767.523,A 0.000,B 0.000,C 90.000,E1 274.245} C_DIS
LIN {X -0.084,Y -342.991,Z 1767.521,A 0.000,B 0.000,C 90.000,E1 273.726} C_DIS
LIN {X -0.097,Y -333.694,Z 1767.517,A 0.000,B 0.000,C 90.000,E1 273.037} C_DIS
LIN {X 0.064,Y -327.169,Z 1767.514,A 0.000,B 0.000,C 90.000,E1 272.579} C_DIS
LIN {X -0.156,Y -320.647,Z 1767.512,A 0.000,B 0.000,C 90.000,E1 272.236} C_DIS
LIN {X 0.146,Y -313.683,Z 1767.510,A 0.000,B 0.000,C 90.000,E1 271.835} C_DIS
LIN {X 0.113,Y -306.482,Z 1767.509,A 0.000,B 0.000,C 90.000,E1 271.547} C_DIS
LIN {X 0.028,Y -299.240,Z 1767.507,A 0.000,B 0.000,C 90.000,E1 271.318} C_DIS
LIN {X 0.044,Y -288.202,Z 1767.506,A 0.000,B 0.000,C 90.000,E1 271.031} C_DIS
LIN {X 0.045,Y -276.792,Z 1767.505,A 0.000,B 0.000,C 90.000,E1 270.802} C_DIS
LIN {X -0.038,Y -264.197,Z 1767.503,A 0.000,B 0.000,C 90.000,E1 270.630} C_DIS
LIN {X 0.113,Y -250.810,Z 1767.503,A 0.000,B 0.000,C 90.000,E1 270.458} C_DIS
LIN {X -0.003,Y -236.518,Z 1767.502,A 0.000,B 0.000,C 90.000,E1 270.401} C_DIS
LIN {X -0.038,Y -181.576,Z 1767.502,A 0.000,B 0.000,C 90.000,E1 270.401} C_DIS
LIN {X 0.048,Y -180.905,Z 1767.474,A 0.000,B 0.000,C 90.000,E1 265.298} C_DIS
LIN {X -0.002,Y -180.251,Z 1767.465,A 0.000,B 0.000,C 90.000,E1 263.628} C_DIS
LIN {X 0.017,Y -178.740,Z 1767.441,A 0.000,B 0.000,C 90.000,E1 259.398} C_DIS
LIN {X -0.086,Y -175.788,Z 1767.413,A 0.000,B 0.000,C 90.000,E1 254.338} C_DIS
LIN {X -0.090,Y -171.972,Z 1767.384,A 0.000,B 0.000,C 90.000,E1 249.209} C_DIS
LIN {X -0.052,Y -171.373,Z 1767.380,A 0.000,B 0.000,C 90.000,E1 248.337} C_DIS
LIN {X -0.066,Y -167.620,Z 1767.356,A 0.000,B 0.000,C 90.000,E1 244.024} C_DIS
LIN {X -0.051,Y -166.270,Z 1767.346,A 0.000,B 0.000,C 90.000,E1 242.281} C_DIS
LIN {X -0.055,Y -163.021,Z 1767.327,A 0.000,B 0.000,C 90.000,E1 238.791} C_DIS
LIN {X -0.003,Y -160.948,Z 1767.312,A 0.000,B 0.000,C 90.000,E1 236.135} C_DIS
LIN {X -0.019,Y -157.705,Z 1767.292,A 0.000,B 0.000,C 90.000,E1 232.603} C_DIS
LIN {X 0.044,Y -155.744,Z 1767.277,A 0.000,B 0.000,C 90.000,E1 229.908} C_DIS
LIN {X -0.009,Y -152.001,Z 1767.252,A 0.000,B 0.000,C 90.000,E1 225.445} C_DIS
LIN {X 0.002,Y -150.247,Z 1767.237,A 0.000,B 0.000,C 90.000,E1 222.732} C_DIS
LIN {X 0.035,Y -147.004,Z 1767.212,A 0.000,B 0.000,C 90.000,E1 218.177} C_DIS
LIN {X 0.025,Y -145.588,Z 1767.197,A 0.000,B 0.000,C 90.000,E1 215.438} C_DIS
LIN {X -0.055,Y -142.976,Z 1767.171,A 0.000,B 0.000,C 90.000,E1 210.875} C_DIS
LIN {X 0.072,Y -141.603,Z 1767.151,A 0.000,B 0.000,C 90.000,E1 207.129} C_DIS
LIN {X -0.013,Y -139.424,Z 1767.115,A 0.000,B 0.000,C 90.000,E1 200.663} C_DIS
LIN {X 0.038,Y -139.153,Z 1767.104,A 0.000,B 0.000,C 90.000,E1 198.779} C_DIS
LIN {X 0.060,Y -138.344,Z 1767.058,A 0.000,B 0.000,C 90.000,E1 190.366} C_DIS
LIN {X 0.046,Y -139.484,Z 1767.006,A 0.000,B 0.000,C 90.000,E1 181.031} C_DIS
LIN {X -0.014,Y -141.082,Z 1766.975,A 0.000,B 0.000,C 90.000,E1 175.469} C_DIS
LIN {X -0.060,Y -142.458,Z 1766.959,A 0.000,B 0.000,C 90.000,E1 172.704} C_DIS
LIN {X 0.030,Y -144.701,Z 1766.934,A 0.000,B 0.000,C 90.000,E1 168.049} C_DIS
LIN {X -0.018,Y -147.297,Z 1766.913,A 0.000,B 0.000,C 90.000,E1 164.393} C_DIS
LIN {X -0.003,Y -150.616,Z 1766.888,A 0.000,B 0.000,C 90.000,E1 159.826} C_DIS
LIN {X -0.067,Y -154.092,Z 1766.868,A 0.000,B 0.000,C 90.000,E1 156.230} C_DIS
LIN {X -0.002,Y -157.514,Z 1766.848,A 0.000,B 0.000,C 90.000,E1 152.615} C_DIS
LIN {X -0.057,Y -161.746,Z 1766.828,A 0.000,B 0.000,C 90.000,E1 149.076} C_DIS
LIN {X 0.049,Y -165.939,Z 1766.808,A 0.000,B 0.000,C 90.000,E1 145.515} C_DIS
LIN {X 0.047,Y -170.929,Z 1766.789,A 0.000,B 0.000,C 90.000,E1 142.029} C_DIS
LIN {X -0.033,Y -175.797,Z 1766.770,A 0.000,B 0.000,C 90.000,E1 138.609} C_DIS
LIN {X 0.095,Y -181.405,Z 1766.751,A 0.000,B 0.000,C 90.000,E1 135.162} C_DIS
LIN {X -0.030,Y -186.906,Z 1766.732,A 0.000,B 0.000,C 90.000,E1 131.838} C_DIS
LIN {X -0.078,Y -191.486,Z 1766.719,A 0.000,B 0.000,C 90.000,E1 129.358} C_DIS
LIN {X 0.129,Y -197.347,Z 1766.700,A 0.000,B 0.000,C 90.000,E1 126.011} C_DIS
LIN {X 0.054,Y -200.623,Z 1766.691,A 0.000,B 0.000,C 90.000,E1 124.405} C_DIS
LIN {X -0.035,Y -206.507,Z 1766.673,A 0.000,B 0.000,C 90.000,E1 121.209} C_DIS
LIN {X -0.036,Y -210.664,Z 1766.662,A 0.000,B 0.000,C 90.000,E1 119.155} C_DIS
LIN {X 0.048,Y -210.757,Z 1766.662,A 0.000,B 0.000,C 90.000,E1 119.077} C_DIS
LIN {X 0.032,Y -336.415,Z 1766.662,A 0.000,B 0.000,C 90.000,E1 119.077} C_DIS
LIN {X -0.012,Y -341.745,Z 1766.661,A 0.000,B 0.000,C 90.000,E1 118.949} C_DIS
LIN {X -0.056,Y -344.018,Z 1766.660,A 0.000,B 0.000,C 90.000,E1 118.821} C_DIS
LIN {X 0.093,Y -347.868,Z 1766.658,A 0.000,B 0.000,C 90.000,E1 118.437} C_DIS
LIN {X 0.211,Y -351.311,Z 1766.655,A 0.000,B 0.000,C 90.000,E1 117.897} C_DIS
LIN {X 0.150,Y -366.062,Z 1766.638,A 0.000,B 0.000,C 90.000,E1 114.899} C_DIS
LIN {X -0.004,Y -380.914,Z 1766.624,A 0.000,B 0.000,C 90.000,E1 112.280} C_DIS
LIN {X -0.068,Y -395.524,Z 1766.611,A 0.000,B 0.000,C 90.000,E1 109.993} C_DIS
LIN {X -0.182,Y -411.562,Z 1766.599,A 0.000,B 0.000,C 90.000,E1 107.764} C_DIS
LIN {X -0.014,Y -429.139,Z 1766.586,A 0.000,B 0.000,C 90.000,E1 105.552} C_DIS
LIN {X 0.052,Y -448.031,Z 1766.575,A 0.000,B 0.000,C 90.000,E1 103.411} C_DIS
LIN {X -0.188,Y -467.495,Z 1766.563,A 0.000,B 0.000,C 90.000,E1 101.366} C_DIS
LIN {X 0.230,Y -484.677,Z 1766.553,A 0.000,B 0.000,C 90.000,E1 99.557} C_DIS
LIN {X 0.076,Y -499.234,Z 1766.545,A 0.000,B 0.000,C 90.000,E1 98.106} C_DIS
LIN {X 0.163,Y -508.679,Z 1766.540,A 0.000,B 0.000,C 90.000,E1 97.125} C_DIS
LIN {X 0.105,Y -510.326,Z 1766.538,A 0.000,B 0.000,C 90.000,E1 96.891} C_DIS
LIN {X -0.015,Y -511.364,Z 1766.537,A 0.000,B 0.000,C 90.000,E1 96.663} C_DIS
LIN {X -0.172,Y -512.116,Z 1766.534,A 0.000,B 0.000,C 90.000,E1 96.201} C_DIS
LIN {X 0.184,Y -511.306,Z 1766.532,A 0.000,B 0.000,C 90.000,E1 95.682} C_DIS
LIN {X 0.085,Y -510.240,Z 1766.530,A 0.000,B 0.000,C 90.000,E1 95.454} C_DIS
LIN {X 0.081,Y -501.813,Z 1766.522,A 0.000,B 0.000,C 90.000,E1 94.012} C_DIS
LIN {X -0.001,Y -494.622,Z 1766.516,A 0.000,B 0.000,C 90.000,E1 92.808} C_DIS
LIN {X -0.183,Y -487.023,Z 1766.509,A 0.000,B 0.000,C 90.000,E1 91.604} C_DIS
LIN {X 0.144,Y -476.026,Z 1766.499,A 0.000,B 0.000,C 90.000,E1 89.828} C_DIS
LIN {X 0.168,Y -467.972,Z 1766.492,A 0.000,B 0.000,C 90.000,E1 88.568} C_DIS
LIN {X -0.128,Y -458.011,Z 1766.484,A 0.000,B 0.000,C 90.000,E1 87.078} C_DIS
LIN {X -0.104,Y -447.819,Z 1766.475,A 0.000,B 0.000,C 90.000,E1 85.527} C_DIS
LIN {X 0.223,Y -437.314,Z 1766.466,A 0.000,B 0.000,C 90.000,E1 83.913} C_DIS
LIN {X -0.065,Y -426.712,Z 1766.458,A 0.000,B 0.000,C 90.000,E1 82.356} C_DIS
LIN {X -0.002,Y -409.361,Z 1766.442,A 0.000,B 0.000,C 90.000,E1 79.634} C_DIS
LIN {X -0.148,Y -391.387,Z 1766.425,A 0.000,B 0.000,C 90.000,E1 76.589} C_DIS
LIN {X -0.108,Y -374.520,Z 1766.408,A 0.000,B 0.000,C 90.000,E1 73.433} C_DIS
LIN {X -0.139,Y -362.784,Z 1766.395,A 0.000,B 0.000,C 90.000,E1 71.094} C_DIS
LIN {X -0.180,Y -349.919,Z 1766.380,A 0.000,B 0.000,C 90.000,E1 68.411} C_DIS
LIN {X 0.123,Y -337.510,Z 1766.365,A 0.000,B 0.000,C 90.000,E1 65.613} C_DIS
LIN {X 0.091,Y -326.816,Z 1766.351,A 0.000,B 0.000,C 90.000,E1 63.127} C_DIS
LIN {X -0.063,Y -318.812,Z 1766.340,A 0.000,B 0.000,C 90.000,E1 61.257} C_DIS
LIN {X -0.055,Y -310.521,Z 1766.330,A 0.000,B 0.000,C 90.000,E1 59.331} C_DIS
LIN {X -0.039,Y -301.713,Z 1766.319,A 0.000,B 0.000,C 90.000,E1 57.375} C_DIS
LIN {X -0.117,Y -288.371,Z 1766.302,A 0.000,B 0.000,C 90.000,E1 54.402} C_DIS
LIN {X -0.070,Y -275.564,Z 1766.285,A 0.000,B 0.000,C 90.000,E1 51.331} C_DIS
LIN {X 0.091,Y -263.400,Z 1766.268,A 0.000,B 0.000,C 90.000,E1 48.162} C_DIS
LIN {X 0.039,Y -253.005,Z 1766.252,A 0.000,B 0.000,C 90.000,E1 45.324} C_DIS
LIN {X -0.096,Y -241.711,Z 1766.234,A 0.000,B 0.000,C 90.000,E1 42.081} C_DIS
LIN {X 0.057,Y -232.180,Z 1766.217,A 0.000,B 0.000,C 90.000,E1 39.072} C_DIS
LIN {X 0.056,Y -224.290,Z 1766.202,A 0.000,B 0.000,C 90.000,E1 36.423} C_DIS
LIN {X -0.029,Y -215.836,Z 1766.185,A 0.000,B 0.000,C 90.000,E1 33.372} C_DIS
LIN {X -0.071,Y -208.035,Z 1766.168,A 0.000,B 0.000,C 90.000,E1 30.256} C_DIS
LIN {X 0.018,Y -200.941,Z 1766.150,A 0.000,B 0.000,C 90.000,E1 27.052} C_DIS
LIN {X 0.017,Y -194.601,Z 1766.132,A 0.000,B 0.000,C 90.000,E1 23.823} C_DIS
LIN {X -0.007,Y -189.085,Z 1766.114,A 0.000,B 0.000,C 90.000,E1 20.556} C_DIS
LIN {X 0.060,Y -184.384,Z 1766.096,A 0.000,B 0.000,C 90.000,E1 17.221} C_DIS
LIN {X 0.023,Y -180.631,Z 1766.077,A 0.000,B 0.000,C 90.000,E1 13.883} C_DIS
LIN {X -0.010,Y -177.021,Z 1766.054,A 0.000,B 0.000,C 90.000,E1 9.670} C_DIS
LIN {X 0.068,Y -174.062,Z 1766.025,A 0.000,B 0.000,C 90.000,E1 4.531} C_DIS
LIN {X -0.025,Y -172.538,Z 1765.988,A 0.000,B 0.000,C 90.000,E1 357.822} C_DIS
LIN {X -0.055,Y -172.861,Z 1765.945,A 0.000,B 0.000,C 90.000,E1 350.095} C_DIS
LIN {X 0.056,Y -175.041,Z 1765.907,A 0.000,B 0.000,C 90.000,E1 343.196} C_DIS
LIN {X -0.020,Y -178.151,Z 1765.878,A 0.000,B 0.000,C 90.000,E1 338.103} C_DIS
LIN {X 0.052,Y -181.489,Z 1765.855,A 0.000,B 0.000,C 90.000,E1 333.845} C_DIS
LIN {X -0.018,Y -185.738,Z 1765.831,A 0.000,B 0.000,C 90.000,E1 329.665} C_DIS
LIN {X -0.042,Y -189.997,Z 1765.813,A 0.000,B 0.000,C 90.000,E1 326.342} C_DIS
LIN {X -0.065,Y -195.164,Z 1765.795,A 0.000,B 0.000,C 90.000,E1 323.050} C_DIS
LIN {X -0.054,Y -199.680,Z 1765.781,A 0.000,B 0.000,C 90.000,E1 320.598} C_DIS
LIN {X -0.013,Y -204.939,Z 1765.768,A 0.000,B 0.000,C 90.000,E1 318.162} C_DIS
LIN {X 0.008,Y -211.931,Z 1765.752,A 0.000,B 0.000,C 90.000,E1 315.364} C_DIS
LIN {X 0.083,Y -217.635,Z 1765.741,A 0.000,B 0.000,C 90.000,E1 313.380} C_DIS
LIN {X -0.040,Y -224.171,Z 1765.730,A 0.000,B 0.000,C 90.000,E1 311.472} C_DIS
LIN {X -0.008,Y -230.105,Z 1765.722,A 0.000,B 0.000,C 90.000,E1 309.930} C_DIS
LIN {X 0.129,Y -236.780,Z 1765.713,A 0.000,B 0.000,C 90.000,E1 308.382} C_DIS
LIN {X -0.147,Y -246.163,Z 1765.703,A 0.000,B 0.000,C 90.000,E1 306.583} C_DIS
LIN {X 0.152,Y -258.627,Z 1765.691,A 0.000,B 0.000,C 90.000,E1 304.326} C_DIS
LIN {X -0.099,Y -276.996,Z 1765.675,A 0.000,B 0.000,C 90.000,E1 301.544} C_DIS
LIN {X -0.176,Y -296.969,Z 1765.660,A 0.000,B 0.000,C 90.000,E1 298.821} C_DIS
LIN {X -0.075,Y -315.118,Z 1765.647,A 0.000,B 0.000,C 90.000,E1 296.488} C_DIS
LIN {X -0.121,Y -328.336,Z 1765.638,A 0.000,B 0.000,C 90.000,E1 294.899} C_DIS
LIN {X -0.129,Y -341.433,Z 1765.630,A 0.000,B 0.000,C 90.000,E1 293.334} C_DIS
LIN {X 0.058,Y -354.172,Z 1765.621,A 0.000,B 0.000,C 90.000,E1 291.770} C_DIS
LIN {X 0.109,Y -364.008,Z 1765.614,A 0.000,B 0.000,C 90.000,E1 290.556} C_DIS
LIN {X -0.098,Y -368.697,Z 1765.611,A 0.000,B 0.000,C 90.000,E1 289.993} C_DIS
LIN {X 0.041,Y -375.008,Z 1765.606,A 0.000,B 0.000,C 90.000,E1 289.087} C_DIS
LIN {X -0.122,Y -380.513,Z 1765.601,A 0.000,B 0.000,C 90.000,E1 288.236} C_DIS
LIN {X 0.132,Y -385.031,Z 1765.596,A 0.000,B 0.000,C 90.000,E1 287.330} C_DIS
LIN {X -0.056,Y -388.612,Z 1765.592,A 0.000,B 0.000,C 90.000,E1 286.496} C_DIS
LIN {X 0.125,Y -390.547,Z 1765.588,A 0.000,B 0.000,C 90.000,E1 285.898} C_DIS
LIN {X -0.169,Y -392.123,Z 1765.585,A 0.000,B 0.000,C 90.000,E1 285.371} C_DIS
LIN {X 0.032,Y -393.310,Z 1765.582,A 0.000,B 0.000,C 90.000,E1 284.773} C_DIS
LIN {X 0.142,Y -394.232,Z 1765.579,A 0.000,B 0.000,C 90.000,E1 284.189} C_DIS
LIN {X -0.026,Y -394.713,Z 1765.576,A 0.000,B 0.000,C 90.000,E1 283.647} C_DIS
LIN {X 0.101,Y -394.847,Z 1765.573,A 0.000,B 0.000,C 90.000,E1 283.063} C_DIS
LIN {X -0.152,Y -394.633,Z 1765.569,A 0.000,B 0.000,C 90.000,E1 282.535} C_DIS
LIN {X -0.019,Y -394.034,Z 1765.566,A 0.000,B 0.000,C 90.000,E1 281.951} C_DIS
LIN {X 0.114,Y -393.007,Z 1765.563,A 0.000,B 0.000,C 90.000,E1 281.366} C_DIS
LIN {X -0.143,Y -391.574,Z 1765.560,A 0.000,B 0.000,C 90.000,E1 280.838} C_DIS
LIN {X -0.021,Y -389.713,Z 1765.557,A 0.000,B 0.000,C 90.000,E1 280.254} C_DIS
LIN {X 0.133,Y -386.070,Z 1765.552,A 0.000,B 0.000,C 90.000,E1 279.378} C_DIS
LIN {X -0.160,Y -380.192,Z 1765.546,A 0.000,B 0.000,C 90.000,E1 278.276} C_DIS
LIN {X -0.152,Y -375.432,Z 1765.541,A 0.000,B 0.000,C 90.000,E1 277.409} C_DIS
LIN {X 0.177,Y -369.910,Z 1765.536,A 0.000,B 0.000,C 90.000,E1 276.486} C_DIS
LIN {X 0.109,Y -365.537,Z 1765.533,A 0.000,B 0.000,C 90.000,E1 275.910} C_DIS
LIN {X 0.020,Y -360.533,Z 1765.530,A 0.000,B 0.000,C 90.000,E1 275.334} C_DIS
LIN {X -0.007,Y -354.948,Z 1765.526,A 0.000,B 0.000,C 90.000,E1 274.759} C_DIS
LIN {X 0.161,Y -349.040,Z 1765.523,A 0.000,B 0.000,C 90.000,E1 274.188} C_DIS
LIN {X -0.076,Y -343.017,Z 1765.521,A 0.000,B 0.000,C 90.000,E1 273.726} C_DIS
LIN {X -0.065,Y -333.706,Z 1765.517,A 0.000,B 0.000,C 90.000,E1 273.037} C_DIS
LIN {X 0.138,Y -327.310,Z 1765.514,A 0.000,B 0.000,C 90.000,E1 272.579} C_DIS
LIN {X -0.084,Y -320.774,Z 1765.512,A 0.000,B 0.000,C 90.000,E1 272.236} C_DIS
LIN {X -0.094,Y -313.828,Z 1765.510,A 0.000,B 0.000,C 90.000,E1 271.892} C_DIS
LIN {X -0.130,Y -306.614,Z 1765.509,A 0.000,B 0.000,C 90.000,E1 271.604} C_DIS
LIN {X 0.090,Y -299.344,Z 1765.507,A 0.000,B 0.000,C 90.000,E1 271.318} C_DIS
LIN {X 0.105,Y -288.366,Z 1765.506,A 0.000,B 0.000,C 90.000,E1 271.031} C_DIS
LIN {X 0.115,Y -277.092,Z 1765.505,A 0.000,B 0.000,C 90.000,E1 270.802} C_DIS
LIN {X 0.039,Y -264.633,Z 1765.504,A 0.000,B 0.000,C 90.000,E1 270.630} C_DIS
LIN {X -0.061,Y -251.467,Z 1765.503,A 0.000,B 0.000,C 90.000,E1 270.516} C_DIS
LIN {X 0.072,Y -237.548,Z 1765.502,A 0.000,B 0.000,C 90.000,E1 270.401} C_DIS
LIN {X 0.025,Y -233.177,Z 1765.502,A 0.000,B 0.000,C 90.000,E1 270.401} C_DIS
LIN {X -0.016,Y -181.576,Z 1765.502,A 0.000,B 0.000,C 90.000,E1 270.401} C_DIS
LIN {X -0.037,Y -180.861,Z 1765.472,A 0.000,B 0.000,C 90.000,E1 265.008} C_DIS
LIN {X 0.016,Y -178.974,Z 1765.444,A 0.000,B 0.000,C 90.000,E1 259.926} C_DIS
LIN {X 0.026,Y -177.935,Z 1765.435,A 0.000,B 0.000,C 90.000,E1 258.229} C_DIS
LIN {X 0.041,Y -175.574,Z 1765.411,A 0.000,B 0.000,C 90.000,E1 253.976} C_DIS
LIN {X 0.048,Y -172.301,Z 1765.387,A 0.000,B 0.000,C 90.000,E1 249.699} C_DIS
LIN {X 0.026,Y -171.781,Z 1765.383,A 0.000,B 0.000,C 90.000,E1 248.847} C_DIS
LIN {X -0.002,Y -168.711,Z 1765.363,A 0.000,B 0.000,C 90.000,E1 245.409} C_DIS
LIN {X 0.036,Y -166.775,Z 1765.349,A 0.000,B 0.000,C 90.000,E1 242.794} C_DIS
LIN {X -0.044,Y -162.756,Z 1765.325,A 0.000,B 0.000,C 90.000,E1 238.456} C_DIS
LIN {X -0.068,Y -161.445,Z 1765.315,A 0.000,B 0.000,C 90.000,E1 236.707} C_DIS
LIN {X -0.026,Y -157.438,Z 1765.290,A 0.000,B 0.000,C 90.000,E1 232.271} C_DIS
LIN {X 0.008,Y -155.446,Z 1765.276,A 0.000,B 0.000,C 90.000,E1 229.585} C_DIS
LIN {X 0.057,Y -151.765,Z 1765.251,A 0.000,B 0.000,C 90.000,E1 225.081} C_DIS
LIN {X 0.068,Y -149.967,Z 1765.235,A 0.000,B 0.000,C 90.000,E1 222.366} C_DIS
LIN {X -0.021,Y -146.806,Z 1765.210,A 0.000,B 0.000,C 90.000,E1 217.855} C_DIS
LIN {X -0.005,Y -145.383,Z 1765.195,A 0.000,B 0.000,C 90.000,E1 215.105} C_DIS
LIN {X -0.013,Y -142.442,Z 1765.164,A 0.000,B 0.000,C 90.000,E1 209.589} C_DIS
LIN {X 0.033,Y -141.434,Z 1765.149,A 0.000,B 0.000,C 90.000,E1 206.796} C_DIS
LIN {X 0.015,Y -139.366,Z 1765.113,A 0.000,B 0.000,C 90.000,E1 200.301} C_DIS
LIN {X 0.001,Y -138.812,Z 1765.097,A 0.000,B 0.000,C 90.000,E1 197.511} C_DIS
LIN {X 0.052,Y -138.351,Z 1765.056,A 0.000,B 0.000,C 90.000,E1 190.018} C_DIS
LIN {X 0.028,Y -139.539,Z 1765.004,A 0.000,B 0.000,C 90.000,E1 180.688} C_DIS
LIN {X -0.020,Y -141.233,Z 1764.973,A 0.000,B 0.000,C 90.000,E1 175.122} C_DIS
LIN {X -0.061,Y -142.604,Z 1764.957,A 0.000,B 0.000,C 90.000,E1 172.356} C_DIS
LIN {X 0.033,Y -144.914,Z 1764.932,A 0.000,B 0.000,C 90.000,E1 167.701} C_DIS
LIN {X 0.026,Y -147.543,Z 1764.911,A 0.000,B 0.000,C 90.000,E1 164.031} C_DIS
LIN {X 0.058,Y -150.143,Z 1764.891,A 0.000,B 0.000,C 90.000,E1 160.369} C_DIS
LIN {X -0.073,Y -153.512,Z 1764.871,A 0.000,B 0.000,C 90.000,E1 156.794} C_DIS
LIN {X -0.011,Y -157.876,Z 1764.846,A 0.000,B 0.000,C 90.000,E1 152.281} C_DIS
LIN {X -0.056,Y -162.163,Z 1764.826,A 0.000,B 0.000,C 90.000,E1 148.742} C_DIS
LIN {X 0.060,Y -166.371,Z 1764.807,A 0.000,B 0.000,C 90.000,E1 145.182} C_DIS
LIN {X 0.062,Y -171.387,Z 1764.787,A 0.000,B 0.000,C 90.000,E1 141.698} C_DIS
LIN {X 0.102,Y -176.298,Z 1764.768,A 0.000,B 0.000,C 90.000,E1 138.243} C_DIS
LIN {X -0.030,Y -180.585,Z 1764.754,A 0.000,B 0.000,C 90.000,E1 135.729} C_DIS
LIN {X -0.051,Y -185.986,Z 1764.735,A 0.000,B 0.000,C 90.000,E1 132.366} C_DIS
LIN {X 0.004,Y -190.620,Z 1764.721,A 0.000,B 0.000,C 90.000,E1 129.850} C_DIS
LIN {X -0.089,Y -196.370,Z 1764.703,A 0.000,B 0.000,C 90.000,E1 126.583} C_DIS
LIN {X -0.012,Y -201.163,Z 1764.690,A 0.000,B 0.000,C 90.000,E1 124.119} C_DIS
LIN {X -0.094,Y -207.107,Z 1764.672,A 0.000,B 0.000,C 90.000,E1 120.924} C_DIS
LIN {X 0.112,Y -210.728,Z 1764.662,A 0.000,B 0.000,C 90.000,E1 119.077} C_DIS
LIN {X 0.133,Y -337.223,Z 1764.662,A 0.000,B 0.000,C 90.000,E1 119.077} C_DIS
LIN {X -0.009,Y -338.662,Z 1764.661,A 0.000,B 0.000,C 90.000,E1 119.077} C_DIS
LIN {X -0.160,Y -344.431,Z 1764.660,A 0.000,B 0.000,C 90.000,E1 118.821} C_DIS
LIN {X 0.160,Y -347.410,Z 1764.658,A 0.000,B 0.000,C 90.000,E1 118.487} C_DIS
LIN {X 0.087,Y -351.004,Z 1764.656,A 0.000,B 0.000,C 90.000,E1 117.975} C_DIS
LIN {X 0.020,Y -365.748,Z 1764.639,A 0.000,B 0.000,C 90.000,E1 114.975} C_DIS
LIN {X 0.004,Y -380.565,Z 1764.624,A 0.000,B 0.000,C 90.000,E1 112.333} C_DIS
LIN {X -0.209,Y -395.143,Z 1764.611,A 0.000,B 0.000,C 90.000,E1 110.066} C_DIS
LIN {X -0.203,Y -411.146,Z 1764.599,A 0.000,B 0.000,C 90.000,E1 107.819} C_DIS
LIN {X -0.052,Y -428.685,Z 1764.587,A 0.000,B 0.000,C 90.000,E1 105.607} C_DIS
LIN {X -0.160,Y -455.307,Z 1764.570,A 0.000,B 0.000,C 90.000,E1 102.703} C_DIS
LIN {X 0.030,Y -475.249,Z 1764.559,A 0.000,B 0.000,C 90.000,E1 100.658} C_DIS
LIN {X -0.052,Y -492.662,Z 1764.550,A 0.000,B 0.000,C 90.000,E1 98.973} C_DIS
LIN {X 0.178,Y -507.451,Z 1764.542,A 0.000,B 0.000,C 90.000,E1 97.530} C_DIS
LIN {X 0.184,Y -509.824,Z 1764.541,A 0.000,B 0.000,C 90.000,E1 97.296} C_DIS
LIN {X 0.095,Y -511.579,Z 1764.539,A 0.000,B 0.000,C 90.000,E1 97.068} C_DIS
LIN {X 0.069,Y -512.774,Z 1764.538,A 0.000,B 0.000,C 90.000,E1 96.834} C_DIS
LIN {X -0.084,Y -513.957,Z 1764.535,A 0.000,B 0.000,C 90.000,E1 96.372} C_DIS
LIN {X -0.231,Y -513.769,Z 1764.533,A 0.000,B 0.000,C 90.000,E1 95.910} C_DIS
LIN {X 0.139,Y -512.161,Z 1764.530,A 0.000,B 0.000,C 90.000,E1 95.391} C_DIS
LIN {X 0.122,Y -503.331,Z 1764.522,A 0.000,B 0.000,C 90.000,E1 93.955} C_DIS
LIN {X -0.070,Y -494.292,Z 1764.514,A 0.000,B 0.000,C 90.000,E1 92.522} C_DIS
LIN {X 0.232,Y -486.359,Z 1764.507,A 0.000,B 0.000,C 90.000,E1 91.260} C_DIS
LIN {X 0.061,Y -474.985,Z 1764.497,A 0.000,B 0.000,C 90.000,E1 89.542} C_DIS
LIN {X -0.112,Y -464.939,Z 1764.489,A 0.000,B 0.000,C 90.000,E1 88.051} C_DIS
LIN {X 0.010,Y -454.635,Z 1764.481,A 0.000,B 0.000,C 90.000,E1 86.502} C_DIS
LIN {X -0.025,Y -444.054,Z 1764.472,A 0.000,B 0.000,C 90.000,E1 84.951} C_DIS
LIN {X 0.134,Y -429.639,Z 1764.460,A 0.000,B 0.000,C 90.000,E1 82.818} C_DIS
LIN {X -0.127,Y -412.126,Z 1764.445,A 0.000,B 0.000,C 90.000,E1 80.151} C_DIS
LIN {X 0.053,Y -395.538,Z 1764.430,A 0.000,B 0.000,C 90.000,E1 77.353} C_DIS
LIN {X 0.115,Y -378.372,Z 1764.412,A 0.000,B 0.000,C 90.000,E1 74.212} C_DIS
LIN {X 0.054,Y -366.486,Z 1764.399,A 0.000,B 0.000,C 90.000,E1 71.891} C_DIS
LIN {X 0.046,Y -354.925,Z 1764.386,A 0.000,B 0.000,C 90.000,E1 69.518} C_DIS
LIN {X 0.048,Y -340.913,Z 1764.369,A 0.000,B 0.000,C 90.000,E1 66.485} C_DIS
LIN {X -0.040,Y -330.125,Z 1764.356,A 0.000,B 0.000,C 90.000,E1 64.024} C_DIS
LIN {X -0.034,Y -320.835,Z 1764.343,A 0.000,B 0.000,C 90.000,E1 61.820} C_DIS
LIN {X 0.134,Y -312.618,Z 1764.333,A 0.000,B 0.000,C 90.000,E1 59.871} C_DIS
LIN {X -0.064,Y -306.930,Z 1764.326,A 0.000,B 0.000,C 90.000,E1 58.614} C_DIS
LIN {X 0.042,Y -298.016,Z 1764.315,A 0.000,B 0.000,C 90.000,E1 56.628} C_DIS
LIN {X 0.018,Y -284.847,Z 1764.298,A 0.000,B 0.000,C 90.000,E1 53.623} C_DIS
LIN {X -0.077,Y -272.206,Z 1764.281,A 0.000,B 0.000,C 90.000,E1 50.561} C_DIS
LIN {X -0.008,Y -260.154,Z 1764.263,A 0.000,B 0.000,C 90.000,E1 47.391} C_DIS
LIN {X 0.027,Y -251.092,Z 1764.249,A 0.000,B 0.000,C 90.000,E1 44.879} C_DIS
LIN {X 0.008,Y -239.887,Z 1764.231,A 0.000,B 0.000,C 90.000,E1 41.595} C_DIS
LIN {X -0.040,Y -230.405,Z 1764.214,A 0.000,B 0.000,C 90.000,E1 38.624} C_DIS
LIN {X -0.030,Y -222.585,Z 1764.200,A 0.000,B 0.000,C 90.000,E1 35.964} C_DIS
LIN {X -0.028,Y -214.228,Z 1764.183,A 0.000,B 0.000,C 90.000,E1 32.880} C_DIS
LIN {X -0.040,Y -206.532,Z 1764.165,A 0.000,B 0.000,C 90.000,E1 29.745} C_DIS
LIN {X 0.015,Y -199.604,Z 1764.147,A 0.000,B 0.000,C 90.000,E1 26.539} C_DIS
LIN {X -0.098,Y -193.401,Z 1764.130,A 0.000,B 0.000,C 90.000,E1 23.334} C_DIS
LIN {X 0.097,Y -188.009,Z 1764.111,A 0.000,B 0.000,C 90.000,E1 19.993} C_DIS
LIN {X 0.074,Y -183.479,Z 1764.093,A 0.000,B 0.000,C 90.000,E1 16.677} C_DIS
LIN {X -0.033,Y -179.866,Z 1764.074,A 0.000,B 0.000,C 90.000,E1 13.355} C_DIS
LIN {X 0.055,Y -176.387,Z 1764.051,A 0.000,B 0.000,C 90.000,E1 9.095} C_DIS
LIN {X -0.059,Y -173.579,Z 1764.022,A 0.000,B 0.000,C 90.000,E1 4.012} C_DIS
LIN {X -0.028,Y -172.302,Z 1763.988,A 0.000,B 0.000,C 90.000,E1 357.822} C_DIS
LIN {X -0.071,Y -172.629,Z 1763.945,A 0.000,B 0.000,C 90.000,E1 350.095} C_DIS
LIN {X 0.028,Y -174.803,Z 1763.907,A 0.000,B 0.000,C 90.000,E1 343.196} C_DIS
LIN {X -0.057,Y -177.924,Z 1763.878,A 0.000,B 0.000,C 90.000,E1 338.103} C_DIS
LIN {X 0.007,Y -181.298,Z 1763.855,A 0.000,B 0.000,C 90.000,E1 333.845} C_DIS
LIN {X -0.069,Y -185.600,Z 1763.831,A 0.000,B 0.000,C 90.000,E1 329.665} C_DIS
LIN {X 0.060,Y -189.890,Z 1763.813,A 0.000,B 0.000,C 90.000,E1 326.294} C_DIS
LIN {X 0.032,Y -195.134,Z 1763.795,A 0.000,B 0.000,C 90.000,E1 323.004} C_DIS
LIN {X 0.011,Y -199.690,Z 1763.781,A 0.000,B 0.000,C 90.000,E1 320.561} C_DIS
LIN {X -0.077,Y -204.995,Z 1763.767,A 0.000,B 0.000,C 90.000,E1 318.162} C_DIS
LIN {X 0.099,Y -212.031,Z 1763.752,A 0.000,B 0.000,C 90.000,E1 315.324} C_DIS
LIN {X 0.026,Y -217.781,Z 1763.741,A 0.000,B 0.000,C 90.000,E1 313.380} C_DIS
LIN {X 0.052,Y -224.353,Z 1763.730,A 0.000,B 0.000,C 90.000,E1 311.434} C_DIS
LIN {X -0.064,Y -230.313,Z 1763.722,A 0.000,B 0.000,C 90.000,E1 309.930} C_DIS
LIN {X 0.075,Y -237.039,Z 1763.713,A 0.000,B 0.000,C 90.000,E1 308.382} C_DIS
LIN {X -0.002,Y -246.455,Z 1763.703,A 0.000,B 0.000,C 90.000,E1 306.537} C_DIS
LIN {X 0.102,Y -258.941,Z 1763.691,A 0.000,B 0.000,C 90.000,E1 304.326} C_DIS
LIN {X 0.002,Y -277.335,Z 1763.675,A 0.000,B 0.000,C 90.000,E1 301.514} C_DIS
LIN {X 0.045,Y -297.331,Z 1763.660,A 0.000,B 0.000,C 90.000,E1 298.771} C_DIS
LIN {X -0.107,Y -315.459,Z 1763.647,A 0.000,B 0.000,C 90.000,E1 296.488} C_DIS
LIN {X 0.087,Y -328.770,Z 1763.638,A 0.000,B 0.000,C 90.000,E1 294.847} C_DIS
LIN {X -0.211,Y -341.840,Z 1763.629,A 0.000,B 0.000,C 90.000,E1 293.334} C_DIS
LIN {X -0.013,Y -354.597,Z 1763.621,A 0.000,B 0.000,C 90.000,E1 291.770} C_DIS
LIN {X 0.041,Y -364.429,Z 1763.614,A 0.000,B 0.000,C 90.000,E1 290.556} C_DIS
LIN {X 0.183,Y -369.098,Z 1763.611,A 0.000,B 0.000,C 90.000,E1 289.939} C_DIS
LIN {X -0.023,Y -375.422,Z 1763.606,A 0.000,B 0.000,C 90.000,E1 289.087} C_DIS
LIN {X 0.179,Y -380.883,Z 1763.601,A 0.000,B 0.000,C 90.000,E1 288.181} C_DIS
LIN {X 0.075,Y -385.416,Z 1763.596,A 0.000,B 0.000,C 90.000,E1 287.330} C_DIS
LIN {X -0.110,Y -388.991,Z 1763.592,A 0.000,B 0.000,C 90.000,E1 286.496} C_DIS
LIN {X 0.073,Y -390.879,Z 1763.588,A 0.000,B 0.000,C 90.000,E1 285.898} C_DIS
LIN {X -0.220,Y -392.501,Z 1763.585,A 0.000,B 0.000,C 90.000,E1 285.371} C_DIS
LIN {X -0.018,Y -393.694,Z 1763.582,A 0.000,B 0.000,C 90.000,E1 284.773} C_DIS
LIN {X 0.096,Y -394.558,Z 1763.579,A 0.000,B 0.000,C 90.000,E1 284.189} C_DIS
LIN {X -0.070,Y -395.034,Z 1763.576,A 0.000,B 0.000,C 90.000,E1 283.647} C_DIS
LIN {X 0.059,Y -395.203,Z 1763.573,A 0.000,B 0.000,C 90.000,E1 283.063} C_DIS
LIN {X -0.193,Y -394.960,Z 1763.569,A 0.000,B 0.000,C 90.000,E1 282.535} C_DIS
LIN {X -0.057,Y -394.341,Z 1763.566,A 0.000,B 0.000,C 90.000,E1 281.951} C_DIS
LIN {X 0.077,Y -393.293,Z 1763.563,A 0.000,B 0.000,C 90.000,E1 281.366} C_DIS
LIN {X -0.177,Y -391.819,Z 1763.560,A 0.000,B 0.000,C 90.000,E1 280.838} C_DIS
LIN {X -0.054,Y -389.868,Z 1763.557,A 0.000,B 0.000,C 90.000,E1 280.254} C_DIS
LIN {X 0.057,Y -387.455,Z 1763.554,A 0.000,B 0.000,C 90.000,E1 279.670} C_DIS
LIN {X 0.159,Y -381.690,Z 1763.547,A 0.000,B 0.000,C 90.000,E1 278.511} C_DIS
LIN {X 0.191,Y -375.442,Z 1763.541,A 0.000,B 0.000,C 90.000,E1 277.352} C_DIS
LIN {X 0.155,Y -371.923,Z 1763.538,A 0.000,B 0.000,C 90.000,E1 276.777} C_DIS
LIN {X 0.100,Y -367.872,Z 1763.535,A 0.000,B 0.000,C 90.000,E1 276.201} C_DIS
LIN {X 0.025,Y -363.186,Z 1763.531,A 0.000,B 0.000,C 90.000,E1 275.625} C_DIS
LIN {X -0.074,Y -357.812,Z 1763.528,A 0.000,B 0.000,C 90.000,E1 275.049} C_DIS
LIN {X -0.010,Y -351.928,Z 1763.525,A 0.000,B 0.000,C 90.000,E1 274.473} C_DIS
LIN {X -0.010,Y -345.985,Z 1763.522,A 0.000,B 0.000,C 90.000,E1 273.955} C_DIS
LIN {X -0.172,Y -339.791,Z 1763.519,A 0.000,B 0.000,C 90.000,E1 273.498} C_DIS
LIN {X 0.057,Y -330.565,Z 1763.516,A 0.000,B 0.000,C 90.000,E1 272.808} C_DIS
LIN {X 0.045,Y -324.082,Z 1763.513,A 0.000,B 0.000,C 90.000,E1 272.407} C_DIS
LIN {X -0.079,Y -317.354,Z 1763.511,A 0.000,B 0.000,C 90.000,E1 272.064} C_DIS
LIN {X 0.059,Y -310.204,Z 1763.510,A 0.000,B 0.000,C 90.000,E1 271.718} C_DIS
LIN {X 0.146,Y -303.003,Z 1763.508,A 0.000,B 0.000,C 90.000,E1 271.432} C_DIS
LIN {X 0.014,Y -292.076,Z 1763.506,A 0.000,B 0.000,C 90.000,E1 271.146} C_DIS
LIN {X -0.052,Y -280.920,Z 1763.505,A 0.000,B 0.000,C 90.000,E1 270.917} C_DIS
LIN {X 0.107,Y -273.112,Z 1763.504,A 0.000,B 0.000,C 90.000,E1 270.745} C_DIS
LIN {X 0.066,Y -259.187,Z 1763.503,A 0.000,B 0.000,C 90.000,E1 270.573} C_DIS
LIN {X 0.014,Y -243.490,Z 1763.503,A 0.000,B 0.000,C 90.000,E1 270.458} C_DIS
LIN {X 0.109,Y -234.605,Z 1763.502,A 0.000,B 0.000,C 90.000,E1 270.401} C_DIS
LIN {X 0.048,Y -181.575,Z 1763.502,A 0.000,B 0.000,C 90.000,E1 270.401} C_DIS
LIN {X -0.046,Y -180.906,Z 1763.474,A 0.000,B 0.000,C 90.000,E1 265.355} C_DIS
LIN {X 0.027,Y -180.674,Z 1763.469,A 0.000,B 0.000,C 90.000,E1 264.489} C_DIS
LIN {X -0.073,Y -178.756,Z 1763.441,A 0.000,B 0.000,C 90.000,E1 259.454} C_DIS
LIN {X 0.000,Y -175.804,Z 1763.413,A 0.000,B 0.000,C 90.000,E1 254.338} C_DIS
LIN {X -0.007,Y -171.989,Z 1763.385,A 0.000,B 0.000,C 90.000,E1 249.209} C_DIS
LIN {X 0.031,Y -171.398,Z 1763.380,A 0.000,B 0.000,C 90.000,E1 248.337} C_DIS
LIN {X 0.016,Y -167.640,Z 1763.356,A 0.000,B 0.000,C 90.000,E1 244.024} C_DIS
LIN {X 0.031,Y -166.299,Z 1763.346,A 0.000,B 0.000,C 90.000,E1 242.281} C_DIS
LIN {X 0.025,Y -163.045,Z 1763.327,A 0.000,B 0.000,C 90.000,E1 238.791} C_DIS
LIN {X -0.013,Y -160.978,Z 1763.312,A 0.000,B 0.000,C 90.000,E1 236.167} C_DIS
LIN {X -0.036,Y -157.728,Z 1763.292,A 0.000,B 0.000,C 90.000,E1 232.637} C_DIS
LIN {X -0.097,Y -155.767,Z 1763.277,A 0.000,B 0.000,C 90.000,E1 229.989} C_DIS
LIN {X -0.041,Y -152.022,Z 1763.253,A 0.000,B 0.000,C 90.000,E1 225.486} C_DIS
LIN {X -0.024,Y -150.269,Z 1763.238,A 0.000,B 0.000,C 90.000,E1 222.771} C_DIS
LIN {X -0.005,Y -147.022,Z 1763.212,A 0.000,B 0.000,C 90.000,E1 218.222} C_DIS
LIN {X 0.016,Y -145.604,Z 1763.197,A 0.000,B 0.000,C 90.000,E1 215.471} C_DIS
LIN {X 0.020,Y -142.990,Z 1763.172,A 0.000,B 0.000,C 90.000,E1 210.875} C_DIS
LIN {X 0.020,Y -141.617,Z 1763.151,A 0.000,B 0.000,C 90.000,E1 207.180} C_DIS
LIN {X 0.060,Y -139.430,Z 1763.115,A 0.000,B 0.000,C 90.000,E1 200.663} C_DIS
LIN {X -0.020,Y -139.160,Z 1763.105,A 0.000,B 0.000,C 90.000,E1 198.833} C_DIS
LIN {X -0.003,Y -138.342,Z 1763.058,A 0.000,B 0.000,C 90.000,E1 190.423} C_DIS
LIN {X -0.021,Y -139.480,Z 1763.006,A 0.000,B 0.000,C 90.000,E1 181.088} C_DIS
LIN {X 0.060,Y -141.069,Z 1762.975,A 0.000,B 0.000,C 90.000,E1 175.469} C_DIS
LIN {X 0.015,Y -142.443,Z 1762.959,A 0.000,B 0.000,C 90.000,E1 172.704} C_DIS
LIN {X -0.037,Y -144.683,Z 1762.934,A 0.000,B 0.000,C 90.000,E1 168.105} C_DIS
LIN {X 0.058,Y -147.273,Z 1762.913,A 0.000,B 0.000,C 90.000,E1 164.393} C_DIS
LIN {X -0.067,Y -150.592,Z 1762.888,A 0.000,B 0.000,C 90.000,E1 159.880} C_DIS
LIN {X 0.011,Y -154.064,Z 1762.868,A 0.000,B 0.000,C 90.000,E1 156.230} C_DIS
LIN {X 0.077,Y -157.483,Z 1762.848,A 0.000,B 0.000,C 90.000,E1 152.615} C_DIS
LIN {X 0.024,Y -161.708,Z 1762.828,A 0.000,B 0.000,C 90.000,E1 149.076} C_DIS
LIN {X 0.037,Y -165.902,Z 1762.809,A 0.000,B 0.000,C 90.000,E1 145.548} C_DIS
LIN {X 0.025,Y -170.886,Z 1762.789,A 0.000,B 0.000,C 90.000,E1 142.065} C_DIS
LIN {X 0.052,Y -175.755,Z 1762.770,A 0.000,B 0.000,C 90.000,E1 138.609} C_DIS
LIN {X -0.075,Y -181.364,Z 1762.751,A 0.000,B 0.000,C 90.000,E1 135.243} C_DIS
LIN {X 0.058,Y -186.858,Z 1762.733,A 0.000,B 0.000,C 90.000,E1 131.838} C_DIS
LIN {X 0.012,Y -191.443,Z 1762.719,A 0.000,B 0.000,C 90.000,E1 129.358} C_DIS
LIN {X -0.056,Y -197.295,Z 1762.700,A 0.000,B 0.000,C 90.000,E1 126.091} C_DIS
LIN {X -0.020,Y -200.573,Z 1762.691,A 0.000,B 0.000,C 90.000,E1 124.452} C_DIS
LIN {X 0.058,Y -206.455,Z 1762.673,A 0.000,B 0.000,C 90.000,E1 121.209} C_DIS
LIN {X 0.013,Y -210.688,Z 1762.662,A 0.000,B 0.000,C 90.000,E1 119.127} C_DIS
LIN {X -0.022,Y -337.064,Z 1762.662,A 0.000,B 0.000,C 90.000,E1 119.127} C_DIS
LIN {X 0.185,Y -338.082,Z 1762.662,A 0.000,B 0.000,C 90.000,E1 119.077} C_DIS
LIN {X 0.097,Y -344.056,Z 1762.660,A 0.000,B 0.000,C 90.000,E1 118.821} C_DIS
LIN {X -0.050,Y -347.110,Z 1762.659,A 0.000,B 0.000,C 90.000,E1 118.565} C_DIS
LIN {X 0.105,Y -350.711,Z 1762.656,A 0.000,B 0.000,C 90.000,E1 118.025} C_DIS
LIN {X 0.095,Y -367.013,Z 1762.637,A 0.000,B 0.000,C 90.000,E1 114.719} C_DIS
LIN {X 0.109,Y -381.983,Z 1762.623,A 0.000,B 0.000,C 90.000,E1 112.078} C_DIS
LIN {X -0.072,Y -396.703,Z 1762.610,A 0.000,B 0.000,C 90.000,E1 109.812} C_DIS
LIN {X -0.156,Y -412.860,Z 1762.598,A 0.000,B 0.000,C 90.000,E1 107.583} C_DIS
LIN {X 0.045,Y -430.565,Z 1762.585,A 0.000,B 0.000,C 90.000,E1 105.371} C_DIS
LIN {X 0.099,Y -449.870,Z 1762.574,A 0.000,B 0.000,C 90.000,E1 103.244} C_DIS
LIN {X 0.081,Y -469.951,Z 1762.563,A 0.000,B 0.000,C 90.000,E1 101.243} C_DIS
LIN {X 0.130,Y -490.155,Z 1762.552,A 0.000,B 0.000,C 90.000,E1 99.321} C_DIS
LIN {X 0.189,Y -507.753,Z 1762.543,A 0.000,B 0.000,C 90.000,E1 97.701} C_DIS
LIN {X 0.187,Y -510.223,Z 1762.542,A 0.000,B 0.000,C 90.000,E1 97.473} C_DIS
LIN {X 0.247,Y -512.132,Z 1762.540,A 0.000,B 0.000,C 90.000,E1 97.239} C_DIS
LIN {X -0.267,Y -513.497,Z 1762.539,A 0.000,B 0.000,C 90.000,E1 97.068} C_DIS
LIN {X 0.096,Y -515.134,Z 1762.536,A 0.000,B 0.000,C 90.000,E1 96.549} C_DIS
LIN {X -0.043,Y -515.464,Z 1762.534,A 0.000,B 0.000,C 90.000,E1 96.087} C_DIS
LIN {X -0.175,Y -514.572,Z 1762.531,A 0.000,B 0.000,C 90.000,E1 95.625} C_DIS
LIN {X -0.216,Y -513.613,Z 1762.530,A 0.000,B 0.000,C 90.000,E1 95.391} C_DIS
LIN {X 0.060,Y -509.157,Z 1762.526,A 0.000,B 0.000,C 90.000,E1 94.645} C_DIS
LIN {X -0.128,Y -498.351,Z 1762.516,A 0.000,B 0.000,C 90.000,E1 92.980} C_DIS
LIN {X 0.234,Y -490.331,Z 1762.510,A 0.000,B 0.000,C 90.000,E1 91.718} C_DIS
LIN {X 0.132,Y -478.686,Z 1762.500,A 0.000,B 0.000,C 90.000,E1 90.000} C_DIS
LIN {X 0.005,Y -468.503,Z 1762.492,A 0.000,B 0.000,C 90.000,E1 88.511} C_DIS
LIN {X 0.178,Y -457.991,Z 1762.483,A 0.000,B 0.000,C 90.000,E1 86.963} C_DIS
LIN {X 0.190,Y -447.227,Z 1762.475,A 0.000,B 0.000,C 90.000,E1 85.412} C_DIS
LIN {X 0.123,Y -430.845,Z 1762.462,A 0.000,B 0.000,C 90.000,E1 83.053} C_DIS
LIN {X -0.112,Y -413.277,Z 1762.447,A 0.000,B 0.000,C 90.000,E1 80.387} C_DIS
LIN {X 0.098,Y -396.598,Z 1762.431,A 0.000,B 0.000,C 90.000,E1 77.589} C_DIS
LIN {X 0.088,Y -379.337,Z 1762.414,A 0.000,B 0.000,C 90.000,E1 74.464} C_DIS
LIN {X 0.153,Y -367.367,Z 1762.401,A 0.000,B 0.000,C 90.000,E1 72.127} C_DIS
LIN {X 0.166,Y -355.752,Z 1762.388,A 0.000,B 0.000,C 90.000,E1 69.752} C_DIS
LIN {X 0.051,Y -343.049,Z 1762.373,A 0.000,B 0.000,C 90.000,E1 67.050} C_DIS
LIN {X 0.014,Y -332.206,Z 1762.359,A 0.000,B 0.000,C 90.000,E1 64.588} C_DIS
LIN {X -0.139,Y -321.551,Z 1762.345,A 0.000,B 0.000,C 90.000,E1 62.103} C_DIS
LIN {X 0.193,Y -313.402,Z 1762.334,A 0.000,B 0.000,C 90.000,E1 60.127} C_DIS
LIN {X 0.052,Y -306.283,Z 1762.325,A 0.000,B 0.000,C 90.000,E1 58.535} C_DIS
LIN {X -0.017,Y -297.393,Z 1762.314,A 0.000,B 0.000,C 90.000,E1 56.580} C_DIS
LIN {X -0.059,Y -284.284,Z 1762.298,A 0.000,B 0.000,C 90.000,E1 53.577} C_DIS
LIN {X -0.007,Y -271.635,Z 1762.280,A 0.000,B 0.000,C 90.000,E1 50.481} C_DIS
LIN {X -0.005,Y -260.918,Z 1762.265,A 0.000,B 0.000,C 90.000,E1 47.676} C_DIS
LIN {X 0.053,Y -251.809,Z 1762.251,A 0.000,B 0.000,C 90.000,E1 45.162} C_DIS
LIN {X -0.116,Y -240.558,Z 1762.233,A 0.000,B 0.000,C 90.000,E1 41.919} C_DIS
LIN {X 0.006,Y -230.997,Z 1762.216,A 0.000,B 0.000,C 90.000,E1 38.910} C_DIS
LIN {X -0.104,Y -220.911,Z 1762.197,A 0.000,B 0.000,C 90.000,E1 35.518} C_DIS
LIN {X -0.082,Y -212.682,Z 1762.180,A 0.000,B 0.000,C 90.000,E1 32.418} C_DIS
LIN {X -0.026,Y -205.160,Z 1762.162,A 0.000,B 0.000,C 90.000,E1 29.255} C_DIS
LIN {X -0.017,Y -198.319,Z 1762.145,A 0.000,B 0.000,C 90.000,E1 26.052} C_DIS
LIN {X -0.075,Y -192.263,Z 1762.127,A 0.000,B 0.000,C 90.000,E1 22.823} C_DIS
LIN {X 0.018,Y -187.003,Z 1762.108,A 0.000,B 0.000,C 90.000,E1 19.504} C_DIS
LIN {X -0.082,Y -182.624,Z 1762.090,A 0.000,B 0.000,C 90.000,E1 16.205} C_DIS
LIN {X -0.029,Y -179.156,Z 1762.071,A 0.000,B 0.000,C 90.000,E1 12.827} C_DIS
LIN {X 0.035,Y -175.818,Z 1762.048,A 0.000,B 0.000,C 90.000,E1 8.568} C_DIS
LIN {X 0.035,Y -173.143,Z 1762.019,A 0.000,B 0.000,C 90.000,E1 3.440} C_DIS
LIN {X -0.031,Y -172.071,Z 1761.988,A 0.000,B 0.000,C 90.000,E1 357.822} C_DIS
LIN {X -0.037,Y -172.580,Z 1761.940,A 0.000,B 0.000,C 90.000,E1 349.218} C_DIS
LIN {X -0.066,Y -175.001,Z 1761.902,A 0.000,B 0.000,C 90.000,E1 342.362} C_DIS
LIN {X -0.024,Y -178.348,Z 1761.873,A 0.000,B 0.000,C 90.000,E1 337.230} C_DIS
LIN {X -0.031,Y -181.892,Z 1761.850,A 0.000,B 0.000,C 90.000,E1 332.999} C_DIS
LIN {X 0.007,Y -186.462,Z 1761.827,A 0.000,B 0.000,C 90.000,E1 328.791} C_DIS
LIN {X -0.001,Y -191.044,Z 1761.808,A 0.000,B 0.000,C 90.000,E1 325.468} C_DIS
LIN {X -0.045,Y -196.561,Z 1761.790,A 0.000,B 0.000,C 90.000,E1 322.190} C_DIS
LIN {X -0.036,Y -201.387,Z 1761.776,A 0.000,B 0.000,C 90.000,E1 319.747} C_DIS
LIN {X -0.060,Y -208.981,Z 1761.758,A 0.000,B 0.000,C 90.000,E1 316.539} C_DIS
LIN {X 0.121,Y -214.370,Z 1761.747,A 0.000,B 0.000,C 90.000,E1 314.514} C_DIS
LIN {X -0.067,Y -220.473,Z 1761.737,A 0.000,B 0.000,C 90.000,E1 312.609} C_DIS
LIN {X -0.084,Y -225.967,Z 1761.728,A 0.000,B 0.000,C 90.000,E1 311.067} C_DIS
LIN {X -0.003,Y -232.150,Z 1761.720,A 0.000,B 0.000,C 90.000,E1 309.519} C_DIS
LIN {X -0.021,Y -239.107,Z 1761.711,A 0.000,B 0.000,C 90.000,E1 308.016} C_DIS
LIN {X -0.062,Y -248.733,Z 1761.701,A 0.000,B 0.000,C 90.000,E1 306.171} C_DIS
LIN {X -0.065,Y -261.490,Z 1761.689,A 0.000,B 0.000,C 90.000,E1 303.992} C_DIS
LIN {X 0.132,Y -280.132,Z 1761.673,A 0.000,B 0.000,C 90.000,E1 301.131} C_DIS
LIN {X 0.146,Y -297.680,Z 1761.660,A 0.000,B 0.000,C 90.000,E1 298.743} C_DIS
LIN {X -0.144,Y -315.807,Z 1761.647,A 0.000,B 0.000,C 90.000,E1 296.488} C_DIS
LIN {X 0.155,Y -331.753,Z 1761.636,A 0.000,B 0.000,C 90.000,E1 294.515} C_DIS
LIN {X -0.067,Y -344.710,Z 1761.628,A 0.000,B 0.000,C 90.000,E1 293.003} C_DIS
LIN {X 0.025,Y -357.418,Z 1761.619,A 0.000,B 0.000,C 90.000,E1 291.461} C_DIS
LIN {X 0.116,Y -367.092,Z 1761.613,A 0.000,B 0.000,C 90.000,E1 290.248} C_DIS
LIN {X -0.114,Y -373.675,Z 1761.608,A 0.000,B 0.000,C 90.000,E1 289.396} C_DIS
LIN {X 0.085,Y -377.659,Z 1761.604,A 0.000,B 0.000,C 90.000,E1 288.779} C_DIS
LIN {X 0.190,Y -381.218,Z 1761.601,A 0.000,B 0.000,C 90.000,E1 288.181} C_DIS
LIN {X -0.044,Y -384.333,Z 1761.598,A 0.000,B 0.000,C 90.000,E1 287.638} C_DIS
LIN {X -0.234,Y -388.249,Z 1761.593,A 0.000,B 0.000,C 90.000,E1 286.804} C_DIS
LIN {X 0.092,Y -391.231,Z 1761.588,A 0.000,B 0.000,C 90.000,E1 285.898} C_DIS
LIN {X -0.198,Y -392.829,Z 1761.585,A 0.000,B 0.000,C 90.000,E1 285.371} C_DIS
LIN {X 0.007,Y -394.032,Z 1761.582,A 0.000,B 0.000,C 90.000,E1 284.773} C_DIS
LIN {X 0.122,Y -394.892,Z 1761.579,A 0.000,B 0.000,C 90.000,E1 284.189} C_DIS
LIN {X -0.042,Y -395.385,Z 1761.576,A 0.000,B 0.000,C 90.000,E1 283.647} C_DIS
LIN {X 0.089,Y -395.500,Z 1761.573,A 0.000,B 0.000,C 90.000,E1 283.063} C_DIS
LIN {X -0.161,Y -395.316,Z 1761.569,A 0.000,B 0.000,C 90.000,E1 282.535} C_DIS
LIN {X -0.023,Y -394.695,Z 1761.566,A 0.000,B 0.000,C 90.000,E1 281.951} C_DIS
LIN {X 0.114,Y -393.617,Z 1761.563,A 0.000,B 0.000,C 90.000,E1 281.366} C_DIS
LIN {X -0.139,Y -392.101,Z 1761.560,A 0.000,B 0.000,C 90.000,E1 280.838} C_DIS
LIN {X -0.014,Y -390.057,Z 1761.557,A 0.000,B 0.000,C 90.000,E1 280.254} C_DIS
LIN {X 0.145,Y -386.188,Z 1761.552,A 0.000,B 0.000,C 90.000,E1 279.378} C_DIS
LIN {X -0.157,Y -377.136,Z 1761.543,A 0.000,B 0.000,C 90.000,E1 277.701} C_DIS
LIN {X -0.173,Y -372.042,Z 1761.538,A 0.000,B 0.000,C 90.000,E1 276.834} C_DIS
LIN {X 0.142,Y -367.989,Z 1761.535,A 0.000,B 0.000,C 90.000,E1 276.201} C_DIS
LIN {X 0.068,Y -363.332,Z 1761.531,A 0.000,B 0.000,C 90.000,E1 275.625} C_DIS
LIN {X -0.031,Y -357.937,Z 1761.528,A 0.000,B 0.000,C 90.000,E1 275.049} C_DIS
LIN {X 0.066,Y -352.090,Z 1761.525,A 0.000,B 0.000,C 90.000,E1 274.473} C_DIS
LIN {X 0.069,Y -346.165,Z 1761.522,A 0.000,B 0.000,C 90.000,E1 273.955} C_DIS
LIN {X -0.122,Y -339.902,Z 1761.519,A 0.000,B 0.000,C 90.000,E1 273.498} C_DIS
LIN {X -0.029,Y -333.634,Z 1761.517,A 0.000,B 0.000,C 90.000,E1 273.037} C_DIS
LIN {X -0.087,Y -327.384,Z 1761.515,A 0.000,B 0.000,C 90.000,E1 272.636} C_DIS
LIN {X -0.015,Y -320.767,Z 1761.512,A 0.000,B 0.000,C 90.000,E1 272.236} C_DIS
LIN {X -0.047,Y -313.627,Z 1761.510,A 0.000,B 0.000,C 90.000,E1 271.892} C_DIS
LIN {X -0.052,Y -306.515,Z 1761.509,A 0.000,B 0.000,C 90.000,E1 271.604} C_DIS
LIN {X -0.065,Y -299.484,Z 1761.508,A 0.000,B 0.000,C 90.000,E1 271.375} C_DIS
LIN {X -0.045,Y -288.662,Z 1761.506,A 0.000,B 0.000,C 90.000,E1 271.088} C_DIS
LIN {X -0.093,Y -276.818,Z 1761.505,A 0.000,B 0.000,C 90.000,E1 270.859} C_DIS
LIN {X 0.099,Y -263.447,Z 1761.504,A 0.000,B 0.000,C 90.000,E1 270.630} C_DIS
LIN {X -0.095,Y -245.952,Z 1761.503,A 0.000,B 0.000,C 90.000,E1 270.516} C_DIS
LIN {X -0.042,Y -237.662,Z 1761.502,A 0.000,B 0.000,C 90.000,E1 270.458} C_DIS
LIN {X -0.068,Y -181.572,Z 1761.502,A 0.000,B 0.000,C 90.000,E1 270.458} C_DIS
LIN {X -0.015,Y -180.905,Z 1761.474,A 0.000,B 0.000,C 90.000,E1 265.355} C_DIS
LIN {X 0.058,Y -180.680,Z 1761.469,A 0.000,B 0.000,C 90.000,E1 264.489} C_DIS
LIN {X -0.043,Y -178.762,Z 1761.441,A 0.000,B 0.000,C 90.000,E1 259.454} C_DIS
LIN {X 0.029,Y -175.809,Z 1761.413,A 0.000,B 0.000,C 90.000,E1 254.338} C_DIS
LIN {X 0.023,Y -171.995,Z 1761.385,A 0.000,B 0.000,C 90.000,E1 249.209} C_DIS
LIN {X -0.002,Y -171.407,Z 1761.380,A 0.000,B 0.000,C 90.000,E1 248.358} C_DIS
LIN {X 0.046,Y -167.648,Z 1761.356,A 0.000,B 0.000,C 90.000,E1 244.024} C_DIS
LIN {X 0.060,Y -166.310,Z 1761.346,A 0.000,B 0.000,C 90.000,E1 242.281} C_DIS
LIN {X 0.054,Y -163.053,Z 1761.327,A 0.000,B 0.000,C 90.000,E1 238.791} C_DIS
LIN {X 0.015,Y -160.987,Z 1761.312,A 0.000,B 0.000,C 90.000,E1 236.167} C_DIS
LIN {X -0.007,Y -157.736,Z 1761.292,A 0.000,B 0.000,C 90.000,E1 232.637} C_DIS
LIN {X -0.069,Y -155.775,Z 1761.278,A 0.000,B 0.000,C 90.000,E1 229.989} C_DIS
LIN {X -0.013,Y -152.029,Z 1761.253,A 0.000,B 0.000,C 90.000,E1 225.486} C_DIS
LIN {X 0.004,Y -150.278,Z 1761.238,A 0.000,B 0.000,C 90.000,E1 222.771} C_DIS
LIN {X 0.022,Y -147.028,Z 1761.212,A 0.000,B 0.000,C 90.000,E1 218.222} C_DIS
LIN {X -0.076,Y -145.610,Z 1761.197,A 0.000,B 0.000,C 90.000,E1 215.518} C_DIS
LIN {X 0.046,Y -142.995,Z 1761.172,A 0.000,B 0.000,C 90.000,E1 210.875} C_DIS
LIN {X -0.019,Y -141.622,Z 1761.151,A 0.000,B 0.000,C 90.000,E1 207.206} C_DIS
LIN {X 0.037,Y -139.431,Z 1761.115,A 0.000,B 0.000,C 90.000,E1 200.684} C_DIS
LIN {X -0.040,Y -139.162,Z 1761.105,A 0.000,B 0.000,C 90.000,E1 198.852} C_DIS
LIN {X -0.002,Y -138.341,Z 1761.058,A 0.000,B 0.000,C 90.000,E1 190.433} C_DIS
LIN {X 0.005,Y -139.478,Z 1761.006,A 0.000,B 0.000,C 90.000,E1 181.088} C_DIS
LIN {X -0.054,Y -141.064,Z 1760.975,A 0.000,B 0.000,C 90.000,E1 175.527} C_DIS
LIN {X 0.041,Y -142.438,Z 1760.960,A 0.000,B 0.000,C 90.000,E1 172.704} C_DIS
LIN {X -0.040,Y -144.676,Z 1760.934,A 0.000,B 0.000,C 90.000,E1 168.117} C_DIS
LIN {X -0.057,Y -147.265,Z 1760.913,A 0.000,B 0.000,C 90.000,E1 164.448} C_DIS
LIN {X -0.039,Y -150.583,Z 1760.888,A 0.000,B 0.000,C 90.000,E1 159.880} C_DIS
LIN {X 0.039,Y -154.054,Z 1760.868,A 0.000,B 0.000,C 90.000,E1 156.230} C_DIS
LIN {X -0.034,Y -157.472,Z 1760.848,A 0.000,B 0.000,C 90.000,E1 152.666} C_DIS
LIN {X 0.053,Y -161.695,Z 1760.828,A 0.000,B 0.000,C 90.000,E1 149.076} C_DIS
LIN {X -0.070,Y -165.889,Z 1760.809,A 0.000,B 0.000,C 90.000,E1 145.595} C_DIS
LIN {X 0.055,Y -170.870,Z 1760.789,A 0.000,B 0.000,C 90.000,E1 142.065} C_DIS
LIN {X -0.034,Y -175.740,Z 1760.770,A 0.000,B 0.000,C 90.000,E1 138.647} C_DIS
LIN {X -0.044,Y -181.350,Z 1760.751,A 0.000,B 0.000,C 90.000,E1 135.243} C_DIS
LIN {X 0.090,Y -186.840,Z 1760.733,A 0.000,B 0.000,C 90.000,E1 131.838} C_DIS
LIN {X 0.043,Y -191.427,Z 1760.719,A 0.000,B 0.000,C 90.000,E1 129.358} C_DIS
LIN {X -0.023,Y -197.277,Z 1760.700,A 0.000,B 0.000,C 90.000,E1 126.091} C_DIS
LIN {X 0.012,Y -200.555,Z 1760.691,A 0.000,B 0.000,C 90.000,E1 124.452} C_DIS
LIN {X -0.086,Y -206.437,Z 1760.674,A 0.000,B 0.000,C 90.000,E1 121.258} C_DIS
LIN {X 0.003,Y -210.646,Z 1760.662,A 0.000,B 0.000,C 90.000,E1 119.155} C_DIS
LIN {X -0.044,Y -336.651,Z 1760.662,A 0.000,B 0.000,C 90.000,E1 119.155} C_DIS
LIN {X -0.014,Y -341.735,Z 1760.661,A 0.000,B 0.000,C 90.000,E1 118.999} C_DIS
LIN {X 0.152,Y -344.098,Z 1760.660,A 0.000,B 0.000,C 90.000,E1 118.821} C_DIS
LIN {X -0.133,Y -347.941,Z 1760.658,A 0.000,B 0.000,C 90.000,E1 118.487} C_DIS
LIN {X 0.146,Y -351.332,Z 1760.655,A 0.000,B 0.000,C 90.000,E1 117.897} C_DIS
LIN {X 0.018,Y -364.494,Z 1760.640,A 0.000,B 0.000,C 90.000,E1 115.207} C_DIS
LIN {X -0.196,Y -379.177,Z 1760.625,A 0.000,B 0.000,C 90.000,E1 112.589} C_DIS
LIN {X 0.060,Y -393.621,Z 1760.613,A 0.000,B 0.000,C 90.000,E1 110.248} C_DIS
LIN {X 0.038,Y -409.481,Z 1760.600,A 0.000,B 0.000,C 90.000,E1 108.000} C_DIS
LIN {X 0.159,Y -426.867,Z 1760.588,A 0.000,B 0.000,C 90.000,E1 105.788} C_DIS
LIN {X 0.187,Y -445.885,Z 1760.576,A 0.000,B 0.000,C 90.000,E1 103.647} C_DIS
LIN {X 0.030,Y -468.427,Z 1760.563,A 0.000,B 0.000,C 90.000,E1 101.422} C_DIS
LIN {X -0.139,Y -488.875,Z 1760.553,A 0.000,B 0.000,C 90.000,E1 99.557} C_DIS
LIN {X 0.181,Y -506.756,Z 1760.544,A 0.000,B 0.000,C 90.000,E1 97.936} C_DIS
LIN {X -0.156,Y -511.625,Z 1760.542,A 0.000,B 0.000,C 90.000,E1 97.530} C_DIS
LIN {X -0.135,Y -513.400,Z 1760.540,A 0.000,B 0.000,C 90.000,E1 97.296} C_DIS
LIN {X -0.178,Y -514.691,Z 1760.539,A 0.000,B 0.000,C 90.000,E1 97.068} C_DIS
LIN {X 0.194,Y -516.240,Z 1760.536,A 0.000,B 0.000,C 90.000,E1 96.549} C_DIS
LIN {X 0.061,Y -516.574,Z 1760.534,A 0.000,B 0.000,C 90.000,E1 96.087} C_DIS
LIN {X -0.065,Y -515.770,Z 1760.531,A 0.000,B 0.000,C 90.000,E1 95.625} C_DIS
LIN {X -0.191,Y -513.655,Z 1760.529,A 0.000,B 0.000,C 90.000,E1 95.163} C_DIS
LIN {X 0.219,Y -502.530,Z 1760.519,A 0.000,B 0.000,C 90.000,E1 93.440} C_DIS
LIN {X 0.150,Y -494.482,Z 1760.513,A 0.000,B 0.000,C 90.000,E1 92.236} C_DIS
LIN {X -0.184,Y -484.340,Z 1760.504,A 0.000,B 0.000,C 90.000,E1 90.802} C_DIS
LIN {X 0.084,Y -472.297,Z 1760.495,A 0.000,B 0.000,C 90.000,E1 89.026} C_DIS
LIN {X -0.138,Y -461.604,Z 1760.486,A 0.000,B 0.000,C 90.000,E1 87.535} C_DIS
LIN {X 0.162,Y -448.859,Z 1760.476,A 0.000,B 0.000,C 90.000,E1 85.698} C_DIS
LIN {X -0.053,Y -434.226,Z 1760.465,A 0.000,B 0.000,C 90.000,E1 83.628} C_DIS
LIN {X 0.080,Y -418.239,Z 1760.451,A 0.000,B 0.000,C 90.000,E1 81.197} C_DIS
LIN {X -0.132,Y -402.946,Z 1760.437,A 0.000,B 0.000,C 90.000,E1 78.757} C_DIS
LIN {X -0.014,Y -385.247,Z 1760.420,A 0.000,B 0.000,C 90.000,E1 75.644} C_DIS
LIN {X 0.091,Y -371.549,Z 1760.406,A 0.000,B 0.000,C 90.000,E1 73.032} C_DIS
LIN {X 0.146,Y -358.319,Z 1760.391,A 0.000,B 0.000,C 90.000,E1 70.369} C_DIS
LIN {X 0.099,Y -345.503,Z 1760.376,A 0.000,B 0.000,C 90.000,E1 67.667} C_DIS
LIN {X -0.034,Y -333.229,Z 1760.361,A 0.000,B 0.000,C 90.000,E1 64.921} C_DIS
LIN {X -0.019,Y -322.517,Z 1760.347,A 0.000,B 0.000,C 90.000,E1 62.410} C_DIS
LIN {X 0.109,Y -315.800,Z 1760.338,A 0.000,B 0.000,C 90.000,E1 60.795} C_DIS
LIN {X 0.005,Y -308.851,Z 1760.329,A 0.000,B 0.000,C 90.000,E1 59.203} C_DIS
LIN {X -0.013,Y -300.046,Z 1760.318,A 0.000,B 0.000,C 90.000,E1 57.248} C_DIS
LIN {X -0.140,Y -286.868,Z 1760.301,A 0.000,B 0.000,C 90.000,E1 54.276} C_DIS
LIN {X 0.032,Y -274.096,Z 1760.284,A 0.000,B 0.000,C 90.000,E1 51.170} C_DIS
LIN {X -0.087,Y -263.266,Z 1760.269,A 0.000,B 0.000,C 90.000,E1 48.405} C_DIS
LIN {X 0.021,Y -254.102,Z 1760.255,A 0.000,B 0.000,C 90.000,E1 45.891} C_DIS
LIN {X 0.080,Y -242.685,Z 1760.237,A 0.000,B 0.000,C 90.000,E1 42.609} C_DIS
LIN {X 0.069,Y -233.010,Z 1760.220,A 0.000,B 0.000,C 90.000,E1 39.644} C_DIS
LIN {X 0.012,Y -222.764,Z 1760.201,A 0.000,B 0.000,C 90.000,E1 36.251} C_DIS
LIN {X 0.007,Y -214.326,Z 1760.184,A 0.000,B 0.000,C 90.000,E1 33.166} C_DIS
LIN {X 0.104,Y -206.649,Z 1760.167,A 0.000,B 0.000,C 90.000,E1 30.001} C_DIS
LIN {X -0.112,Y -199.674,Z 1760.149,A 0.000,B 0.000,C 90.000,E1 26.873} C_DIS
LIN {X 0.042,Y -193.436,Z 1760.131,A 0.000,B 0.000,C 90.000,E1 23.590} C_DIS
LIN {X 0.061,Y -187.990,Z 1760.113,A 0.000,B 0.000,C 90.000,E1 20.301} C_DIS
LIN {X 0.041,Y -183.394,Z 1760.094,A 0.000,B 0.000,C 90.000,E1 16.985} C_DIS
LIN {X -0.019,Y -179.703,Z 1760.076,A 0.000,B 0.000,C 90.000,E1 13.647} C_DIS
LIN {X 0.092,Y -176.177,Z 1760.052,A 0.000,B 0.000,C 90.000,E1 9.378} C_DIS
LIN {X -0.053,Y -173.226,Z 1760.024,A 0.000,B 0.000,C 90.000,E1 4.302} C_DIS
LIN {X -0.034,Y -171.831,Z 1759.988,A 0.000,B 0.000,C 90.000,E1 357.822} C_DIS
LIN {X -0.055,Y -172.343,Z 1759.940,A 0.000,B 0.000,C 90.000,E1 349.218} C_DIS
LIN {X 0.071,Y -174.780,Z 1759.902,A 0.000,B 0.000,C 90.000,E1 342.308} C_DIS
LIN {X -0.062,Y -178.149,Z 1759.873,A 0.000,B 0.000,C 90.000,E1 337.230} C_DIS
LIN {X -0.075,Y -181.728,Z 1759.850,A 0.000,B 0.000,C 90.000,E1 332.999} C_DIS
LIN {X -0.044,Y -186.358,Z 1759.827,A 0.000,B 0.000,C 90.000,E1 328.791} C_DIS
LIN {X -0.056,Y -190.979,Z 1759.808,A 0.000,B 0.000,C 90.000,E1 325.468} C_DIS
LIN {X -0.102,Y -196.555,Z 1759.790,A 0.000,B 0.000,C 90.000,E1 322.190} C_DIS
LIN {X 0.059,Y -201.431,Z 1759.776,A 0.000,B 0.000,C 90.000,E1 319.703} C_DIS
LIN {X 0.025,Y -209.059,Z 1759.758,A 0.000,B 0.000,C 90.000,E1 316.500} C_DIS
LIN {X 0.062,Y -214.500,Z 1759.747,A 0.000,B 0.000,C 90.000,E1 314.514} C_DIS
LIN {X -0.127,Y -220.636,Z 1759.737,A 0.000,B 0.000,C 90.000,E1 312.609} C_DIS
LIN {X 0.113,Y -227.653,Z 1759.726,A 0.000,B 0.000,C 90.000,E1 310.620} C_DIS
LIN {X 0.042,Y -234.088,Z 1759.717,A 0.000,B 0.000,C 90.000,E1 309.116} C_DIS
LIN {X 0.063,Y -243.127,Z 1759.707,A 0.000,B 0.000,C 90.000,E1 307.237} C_DIS
LIN {X 0.102,Y -255.292,Z 1759.695,A 0.000,B 0.000,C 90.000,E1 305.025} C_DIS
LIN {X -0.090,Y -273.284,Z 1759.679,A 0.000,B 0.000,C 90.000,E1 302.212} C_DIS
LIN {X 0.134,Y -292.915,Z 1759.664,A 0.000,B 0.000,C 90.000,E1 299.411} C_DIS
LIN {X -0.114,Y -310.894,Z 1759.651,A 0.000,B 0.000,C 90.000,E1 297.129} C_DIS
LIN {X 0.106,Y -326.732,Z 1759.640,A 0.000,B 0.000,C 90.000,E1 295.155} C_DIS
LIN {X -0.076,Y -339.636,Z 1759.631,A 0.000,B 0.000,C 90.000,E1 293.643} C_DIS
LIN {X 0.092,Y -352.508,Z 1759.623,A 0.000,B 0.000,C 90.000,E1 292.078} C_DIS
LIN {X -0.152,Y -362.381,Z 1759.616,A 0.000,B 0.000,C 90.000,E1 290.918} C_DIS
LIN {X 0.045,Y -369.461,Z 1759.611,A 0.000,B 0.000,C 90.000,E1 289.993} C_DIS
LIN {X 0.193,Y -375.809,Z 1759.606,A 0.000,B 0.000,C 90.000,E1 289.087} C_DIS
LIN {X -0.073,Y -379.612,Z 1759.603,A 0.000,B 0.000,C 90.000,E1 288.544} C_DIS
LIN {X 0.045,Y -382.955,Z 1759.600,A 0.000,B 0.000,C 90.000,E1 287.946} C_DIS
LIN {X -0.180,Y -385.905,Z 1759.597,A 0.000,B 0.000,C 90.000,E1 287.402} C_DIS
LIN {X 0.125,Y -389.548,Z 1759.592,A 0.000,B 0.000,C 90.000,E1 286.496} C_DIS
LIN {X -0.064,Y -391.451,Z 1759.589,A 0.000,B 0.000,C 90.000,E1 285.953} C_DIS
LIN {X 0.025,Y -393.064,Z 1759.585,A 0.000,B 0.000,C 90.000,E1 285.371} C_DIS
LIN {X -0.149,Y -394.285,Z 1759.582,A 0.000,B 0.000,C 90.000,E1 284.828} C_DIS
LIN {X -0.034,Y -395.175,Z 1759.579,A 0.000,B 0.000,C 90.000,E1 284.245} C_DIS
LIN {X 0.186,Y -395.683,Z 1759.576,A 0.000,B 0.000,C 90.000,E1 283.647} C_DIS
LIN {X -0.066,Y -395.859,Z 1759.573,A 0.000,B 0.000,C 90.000,E1 283.119} C_DIS
LIN {X 0.071,Y -395.650,Z 1759.570,A 0.000,B 0.000,C 90.000,E1 282.535} C_DIS
LIN {X -0.176,Y -395.050,Z 1759.567,A 0.000,B 0.000,C 90.000,E1 282.007} C_DIS
LIN {X -0.037,Y -393.989,Z 1759.563,A 0.000,B 0.000,C 90.000,E1 281.422} C_DIS
LIN {X 0.097,Y -392.453,Z 1759.560,A 0.000,B 0.000,C 90.000,E1 280.838} C_DIS
LIN {X -0.161,Y -390.384,Z 1759.557,A 0.000,B 0.000,C 90.000,E1 280.310} C_DIS
LIN {X -0.062,Y -386.444,Z 1759.552,A 0.000,B 0.000,C 90.000,E1 279.443} C_DIS
LIN {X 0.080,Y -377.364,Z 1759.543,A 0.000,B 0.000,C 90.000,E1 277.701} C_DIS
LIN {X 0.061,Y -372.333,Z 1759.538,A 0.000,B 0.000,C 90.000,E1 276.834} C_DIS
LIN {X 0.010,Y -368.342,Z 1759.535,A 0.000,B 0.000,C 90.000,E1 276.258} C_DIS
LIN {X -0.061,Y -363.755,Z 1759.531,A 0.000,B 0.000,C 90.000,E1 275.682} C_DIS
LIN {X -0.157,Y -358.337,Z 1759.528,A 0.000,B 0.000,C 90.000,E1 275.106} C_DIS
LIN {X -0.066,Y -352.529,Z 1759.525,A 0.000,B 0.000,C 90.000,E1 274.531} C_DIS
LIN {X -0.059,Y -346.563,Z 1759.522,A 0.000,B 0.000,C 90.000,E1 274.012} C_DIS
LIN {X 0.112,Y -340.419,Z 1759.520,A 0.000,B 0.000,C 90.000,E1 273.498} C_DIS
LIN {X -0.045,Y -330.967,Z 1759.516,A 0.000,B 0.000,C 90.000,E1 272.865} C_DIS
LIN {X -0.036,Y -324.621,Z 1759.514,A 0.000,B 0.000,C 90.000,E1 272.465} C_DIS
LIN {X -0.154,Y -317.897,Z 1759.512,A 0.000,B 0.000,C 90.000,E1 272.121} C_DIS
LIN {X 0.007,Y -310.979,Z 1759.510,A 0.000,B 0.000,C 90.000,E1 271.776} C_DIS
LIN {X 0.108,Y -303.808,Z 1759.508,A 0.000,B 0.000,C 90.000,E1 271.489} C_DIS
LIN {X -0.074,Y -292.720,Z 1759.507,A 0.000,B 0.000,C 90.000,E1 271.203} C_DIS
LIN {X 0.122,Y -281.692,Z 1759.505,A 0.000,B 0.000,C 90.000,E1 270.917} C_DIS
LIN {X -0.013,Y -273.677,Z 1759.504,A 0.000,B 0.000,C 90.000,E1 270.802} C_DIS
LIN {X -0.038,Y -259.333,Z 1759.503,A 0.000,B 0.000,C 90.000,E1 270.630} C_DIS
LIN {X -0.084,Y -243.938,Z 1759.503,A 0.000,B 0.000,C 90.000,E1 270.516} C_DIS
LIN {X 0.016,Y -237.357,Z 1759.503,A 0.000,B 0.000,C 90.000,E1 270.458} C_DIS
LIN {X -0.024,Y -181.571,Z 1759.503,A 0.000,B 0.000,C 90.000,E1 270.458} C_DIS
LIN {X 0.065,Y -180.906,Z 1759.474,A 0.000,B 0.000,C 90.000,E1 265.355} C_DIS
LIN {X -0.041,Y -180.692,Z 1759.470,A 0.000,B 0.000,C 90.000,E1 264.546} C_DIS
LIN {X 0.036,Y -178.776,Z 1759.442,A 0.000,B 0.000,C 90.000,E1 259.454} C_DIS
LIN {X -0.060,Y -175.823,Z 1759.413,A 0.000,B 0.000,C 90.000,E1 254.393} C_DIS
LIN {X -0.060,Y -172.010,Z 1759.385,A 0.000,B 0.000,C 90.000,E1 249.263} C_DIS
LIN {X -0.083,Y -171.429,Z 1759.380,A 0.000,B 0.000,C 90.000,E1 248.411} C_DIS
LIN {X -0.028,Y -167.666,Z 1759.356,A 0.000,B 0.000,C 90.000,E1 244.076} C_DIS
LIN {X -0.088,Y -166.338,Z 1759.346,A 0.000,B 0.000,C 90.000,E1 242.359} C_DIS
LIN {X -0.095,Y -163.076,Z 1759.327,A 0.000,B 0.000,C 90.000,E1 238.869} C_DIS
LIN {X -0.043,Y -161.015,Z 1759.312,A 0.000,B 0.000,C 90.000,E1 236.215} C_DIS
LIN {X 0.067,Y -157.757,Z 1759.293,A 0.000,B 0.000,C 90.000,E1 232.637} C_DIS
LIN {X 0.004,Y -155.796,Z 1759.278,A 0.000,B 0.000,C 90.000,E1 229.989} C_DIS
LIN {X 0.060,Y -152.049,Z 1759.253,A 0.000,B 0.000,C 90.000,E1 225.486} C_DIS
LIN {X 0.077,Y -150.298,Z 1759.238,A 0.000,B 0.000,C 90.000,E1 222.771} C_DIS
LIN {X 0.002,Y -147.044,Z 1759.213,A 0.000,B 0.000,C 90.000,E1 218.257} C_DIS
LIN {X -0.006,Y -145.624,Z 1759.197,A 0.000,B 0.000,C 90.000,E1 215.518} C_DIS
LIN {X -0.007,Y -143.008,Z 1759.172,A 0.000,B 0.000,C 90.000,E1 210.924} C_DIS
LIN {X -0.076,Y -141.634,Z 1759.151,A 0.000,B 0.000,C 90.000,E1 207.257} C_DIS
LIN {X -0.025,Y -139.437,Z 1759.115,A 0.000,B 0.000,C 90.000,E1 200.737} C_DIS
LIN {X 0.029,Y -139.169,Z 1759.105,A 0.000,B 0.000,C 90.000,E1 198.852} C_DIS
LIN {X 0.063,Y -138.317,Z 1759.053,A 0.000,B 0.000,C 90.000,E1 189.500} C_DIS
LIN {X -0.065,Y -139.475,Z 1759.006,A 0.000,B 0.000,C 90.000,E1 181.146} C_DIS
LIN {X 0.016,Y -141.052,Z 1758.975,A 0.000,B 0.000,C 90.000,E1 175.527} C_DIS
LIN {X -0.030,Y -142.424,Z 1758.960,A 0.000,B 0.000,C 90.000,E1 172.761} C_DIS
LIN {X 0.030,Y -144.660,Z 1758.934,A 0.000,B 0.000,C 90.000,E1 168.117} C_DIS
LIN {X 0.015,Y -147.243,Z 1758.914,A 0.000,B 0.000,C 90.000,E1 164.448} C_DIS
LIN {X 0.033,Y -150.560,Z 1758.888,A 0.000,B 0.000,C 90.000,E1 159.880} C_DIS
LIN {X -0.029,Y -154.027,Z 1758.868,A 0.000,B 0.000,C 90.000,E1 156.282} C_DIS
LIN {X 0.040,Y -157.443,Z 1758.848,A 0.000,B 0.000,C 90.000,E1 152.666} C_DIS
LIN {X -0.011,Y -161.660,Z 1758.828,A 0.000,B 0.000,C 90.000,E1 149.125} C_DIS
LIN {X 0.006,Y -165.855,Z 1758.809,A 0.000,B 0.000,C 90.000,E1 145.595} C_DIS
LIN {X -0.002,Y -170.830,Z 1758.790,A 0.000,B 0.000,C 90.000,E1 142.110} C_DIS
LIN {X 0.046,Y -175.700,Z 1758.770,A 0.000,B 0.000,C 90.000,E1 138.647} C_DIS
LIN {X 0.037,Y -181.312,Z 1758.751,A 0.000,B 0.000,C 90.000,E1 135.243} C_DIS
LIN {X -0.091,Y -186.795,Z 1758.733,A 0.000,B 0.000,C 90.000,E1 131.919} C_DIS
LIN {X -0.021,Y -191.386,Z 1758.719,A 0.000,B 0.000,C 90.000,E1 129.402} C_DIS
LIN {X 0.061,Y -197.229,Z 1758.701,A 0.000,B 0.000,C 90.000,E1 126.091} C_DIS
LIN {X -0.015,Y -200.508,Z 1758.692,A 0.000,B 0.000,C 90.000,E1 124.485} C_DIS
LIN {X 0.002,Y -206.389,Z 1758.674,A 0.000,B 0.000,C 90.000,E1 121.258} C_DIS
LIN {X -0.094,Y -210.606,Z 1758.662,A 0.000,B 0.000,C 90.000,E1 119.205} C_DIS
LIN {X 0.095,Y -336.337,Z 1758.662,A 0.000,B 0.000,C 90.000,E1 119.155} C_DIS
LIN {X -0.037,Y -341.582,Z 1758.661,A 0.000,B 0.000,C 90.000,E1 119.027} C_DIS
LIN {X -0.006,Y -343.953,Z 1758.660,A 0.000,B 0.000,C 90.000,E1 118.871} C_DIS
LIN {X 0.021,Y -347.794,Z 1758.658,A 0.000,B 0.000,C 90.000,E1 118.487} C_DIS
LIN {X -0.168,Y -351.189,Z 1758.655,A 0.000,B 0.000,C 90.000,E1 117.975} C_DIS
LIN {X 0.181,Y -364.339,Z 1758.640,A 0.000,B 0.000,C 90.000,E1 115.207} C_DIS
LIN {X -0.031,Y -379.006,Z 1758.625,A 0.000,B 0.000,C 90.000,E1 112.589} C_DIS
LIN {X -0.143,Y -393.435,Z 1758.613,A 0.000,B 0.000,C 90.000,E1 110.301} C_DIS
LIN {X 0.206,Y -409.279,Z 1758.600,A 0.000,B 0.000,C 90.000,E1 108.000} C_DIS
LIN {X -0.082,Y -426.648,Z 1758.588,A 0.000,B 0.000,C 90.000,E1 105.843} C_DIS
LIN {X -0.076,Y -445.650,Z 1758.576,A 0.000,B 0.000,C 90.000,E1 103.703} C_DIS
LIN {X -0.224,Y -465.648,Z 1758.565,A 0.000,B 0.000,C 90.000,E1 101.715} C_DIS
LIN {X -0.088,Y -488.744,Z 1758.553,A 0.000,B 0.000,C 90.000,E1 99.613} C_DIS
LIN {X 0.172,Y -509.427,Z 1758.544,A 0.000,B 0.000,C 90.000,E1 97.814} C_DIS
LIN {X -0.243,Y -511.817,Z 1758.542,A 0.000,B 0.000,C 90.000,E1 97.644} C_DIS
LIN {X -0.161,Y -513.661,Z 1758.541,A 0.000,B 0.000,C 90.000,E1 97.409} C_DIS
LIN {X -0.146,Y -515.034,Z 1758.540,A 0.000,B 0.000,C 90.000,E1 97.182} C_DIS
LIN {X 0.226,Y -516.823,Z 1758.537,A 0.000,B 0.000,C 90.000,E1 96.663} C_DIS
LIN {X 0.094,Y -517.411,Z 1758.535,A 0.000,B 0.000,C 90.000,E1 96.201} C_DIS
LIN {X -0.030,Y -516.918,Z 1758.532,A 0.000,B 0.000,C 90.000,E1 95.739} C_DIS
LIN {X -0.152,Y -515.255,Z 1758.529,A 0.000,B 0.000,C 90.000,E1 95.277} C_DIS
LIN {X -0.237,Y -513.877,Z 1758.528,A 0.000,B 0.000,C 90.000,E1 95.049} C_DIS
LIN {X 0.094,Y -500.807,Z 1758.517,A 0.000,B 0.000,C 90.000,E1 93.094} C_DIS
LIN {X -0.021,Y -492.469,Z 1758.510,A 0.000,B 0.000,C 90.000,E1 91.892} C_DIS
LIN {X -0.064,Y -480.229,Z 1758.501,A 0.000,B 0.000,C 90.000,E1 90.172} C_DIS
LIN {X -0.161,Y -469.559,Z 1758.493,A 0.000,B 0.000,C 90.000,E1 88.682} C_DIS
LIN {X -0.183,Y -456.712,Z 1758.483,A 0.000,B 0.000,C 90.000,E1 86.906} C_DIS
LIN {X 0.041,Y -443.912,Z 1758.473,A 0.000,B 0.000,C 90.000,E1 85.065} C_DIS
LIN {X -0.098,Y -427.604,Z 1758.459,A 0.000,B 0.000,C 90.000,E1 82.704} C_DIS
LIN {X -0.009,Y -410.173,Z 1758.444,A 0.000,B 0.000,C 90.000,E1 79.982} C_DIS
LIN {X 0.186,Y -393.600,Z 1758.429,A 0.000,B 0.000,C 90.000,E1 77.173} C_DIS
LIN {X 0.047,Y -379.496,Z 1758.415,A 0.000,B 0.000,C 90.000,E1 74.629} C_DIS
LIN {X 0.018,Y -367.435,Z 1758.402,A 0.000,B 0.000,C 90.000,E1 72.308} C_DIS
LIN {X 0.036,Y -355.746,Z 1758.389,A 0.000,B 0.000,C 90.000,E1 69.934} C_DIS
LIN {X -0.058,Y -341.624,Z 1758.372,A 0.000,B 0.000,C 90.000,E1 66.922} C_DIS
LIN {X -0.125,Y -330.775,Z 1758.358,A 0.000,B 0.000,C 90.000,E1 64.460} C_DIS
LIN {X 0.124,Y -320.087,Z 1758.344,A 0.000,B 0.000,C 90.000,E1 61.897} C_DIS
LIN {X -0.064,Y -313.308,Z 1758.335,A 0.000,B 0.000,C 90.000,E1 60.333} C_DIS
LIN {X -0.044,Y -306.222,Z 1758.326,A 0.000,B 0.000,C 90.000,E1 58.712} C_DIS
LIN {X 0.145,Y -297.367,Z 1758.315,A 0.000,B 0.000,C 90.000,E1 56.707} C_DIS
LIN {X -0.040,Y -285.771,Z 1758.300,A 0.000,B 0.000,C 90.000,E1 54.069} C_DIS
LIN {X -0.005,Y -274.403,Z 1758.285,A 0.000,B 0.000,C 90.000,E1 51.331} C_DIS
LIN {X 0.120,Y -262.221,Z 1758.268,A 0.000,B 0.000,C 90.000,E1 48.162} C_DIS
LIN {X 0.018,Y -253.045,Z 1758.254,A 0.000,B 0.000,C 90.000,E1 45.688} C_DIS
LIN {X -0.120,Y -241.657,Z 1758.236,A 0.000,B 0.000,C 90.000,E1 42.447} C_DIS
LIN {X -0.009,Y -230.832,Z 1758.217,A 0.000,B 0.000,C 90.000,E1 39.072} C_DIS
LIN {X 0.010,Y -220.690,Z 1758.198,A 0.000,B 0.000,C 90.000,E1 35.644} C_DIS
LIN {X 0.011,Y -212.413,Z 1758.181,A 0.000,B 0.000,C 90.000,E1 32.546} C_DIS
LIN {X -0.045,Y -204.943,Z 1758.163,A 0.000,B 0.000,C 90.000,E1 29.411} C_DIS
LIN {X 0.057,Y -198.109,Z 1758.146,A 0.000,B 0.000,C 90.000,E1 26.181} C_DIS
LIN {X -0.008,Y -192.044,Z 1758.127,A 0.000,B 0.000,C 90.000,E1 22.950} C_DIS
LIN {X 0.081,Y -186.787,Z 1758.109,A 0.000,B 0.000,C 90.000,E1 19.631} C_DIS
LIN {X 0.029,Y -182.344,Z 1758.091,A 0.000,B 0.000,C 90.000,E1 16.315} C_DIS
LIN {X 0.067,Y -178.853,Z 1758.072,A 0.000,B 0.000,C 90.000,E1 12.939} C_DIS
LIN {X -0.085,Y -175.484,Z 1758.048,A 0.000,B 0.000,C 90.000,E1 8.746} C_DIS
LIN {X -0.074,Y -172.750,Z 1758.020,A 0.000,B 0.000,C 90.000,E1 3.612} C_DIS
LIN {X -0.044,Y -171.521,Z 1757.983,A 0.000,B 0.000,C 90.000,E1 356.963} C_DIS
LIN {X -0.023,Y -172.327,Z 1757.935,A 0.000,B 0.000,C 90.000,E1 348.342} C_DIS
LIN {X 0.043,Y -174.567,Z 1757.902,A 0.000,B 0.000,C 90.000,E1 342.308} C_DIS
LIN {X 0.066,Y -177.949,Z 1757.873,A 0.000,B 0.000,C 90.000,E1 337.177} C_DIS
LIN {X 0.042,Y -181.576,Z 1757.850,A 0.000,B 0.000,C 90.000,E1 332.948} C_DIS
LIN {X 0.067,Y -186.240,Z 1757.826,A 0.000,B 0.000,C 90.000,E1 328.742} C_DIS
LIN {X -0.001,Y -190.919,Z 1757.808,A 0.000,B 0.000,C 90.000,E1 325.435} C_DIS
LIN {X -0.002,Y -196.547,Z 1757.790,A 0.000,B 0.000,C 90.000,E1 322.145} C_DIS
LIN {X 0.001,Y -201.461,Z 1757.776,A 0.000,B 0.000,C 90.000,E1 319.703} C_DIS
LIN {X -0.029,Y -209.145,Z 1757.758,A 0.000,B 0.000,C 90.000,E1 316.500} C_DIS
LIN {X 0.003,Y -214.629,Z 1757.747,A 0.000,B 0.000,C 90.000,E1 314.514} C_DIS
LIN {X 0.126,Y -220.814,Z 1757.736,A 0.000,B 0.000,C 90.000,E1 312.528} C_DIS
LIN {X 0.056,Y -227.877,Z 1757.726,A 0.000,B 0.000,C 90.000,E1 310.620} C_DIS
LIN {X -0.015,Y -234.338,Z 1757.717,A 0.000,B 0.000,C 90.000,E1 309.116} C_DIS
LIN {X 0.008,Y -243.440,Z 1757.707,A 0.000,B 0.000,C 90.000,E1 307.237} C_DIS
LIN {X -0.073,Y -257.771,Z 1757.693,A 0.000,B 0.000,C 90.000,E1 304.692} C_DIS
LIN {X 0.172,Y -276.007,Z 1757.677,A 0.000,B 0.000,C 90.000,E1 301.799} C_DIS
LIN {X 0.082,Y -295.786,Z 1757.662,A 0.000,B 0.000,C 90.000,E1 299.077} C_DIS
LIN {X 0.163,Y -313.828,Z 1757.649,A 0.000,B 0.000,C 90.000,E1 296.744} C_DIS
LIN {X 0.035,Y -329.689,Z 1757.638,A 0.000,B 0.000,C 90.000,E1 294.847} C_DIS
LIN {X -0.063,Y -342.501,Z 1757.630,A 0.000,B 0.000,C 90.000,E1 293.334} C_DIS
LIN {X 0.133,Y -355.353,Z 1757.621,A 0.000,B 0.000,C 90.000,E1 291.770} C_DIS
LIN {X -0.140,Y -365.146,Z 1757.614,A 0.000,B 0.000,C 90.000,E1 290.610} C_DIS
LIN {X 0.003,Y -369.804,Z 1757.611,A 0.000,B 0.000,C 90.000,E1 289.993} C_DIS
LIN {X 0.154,Y -376.152,Z 1757.606,A 0.000,B 0.000,C 90.000,E1 289.087} C_DIS
LIN {X -0.111,Y -379.958,Z 1757.603,A 0.000,B 0.000,C 90.000,E1 288.544} C_DIS
LIN {X 0.009,Y -383.334,Z 1757.600,A 0.000,B 0.000,C 90.000,E1 287.946} C_DIS
LIN {X -0.079,Y -387.583,Z 1757.595,A 0.000,B 0.000,C 90.000,E1 287.094} C_DIS
LIN {X 0.094,Y -389.892,Z 1757.592,A 0.000,B 0.000,C 90.000,E1 286.496} C_DIS
LIN {X -0.093,Y -391.799,Z 1757.589,A 0.000,B 0.000,C 90.000,E1 285.953} C_DIS
LIN {X -0.002,Y -393.375,Z 1757.585,A 0.000,B 0.000,C 90.000,E1 285.371} C_DIS
LIN {X 0.207,Y -394.603,Z 1757.582,A 0.000,B 0.000,C 90.000,E1 284.773} C_DIS
LIN {X -0.058,Y -395.495,Z 1757.579,A 0.000,B 0.000,C 90.000,E1 284.245} C_DIS
LIN {X 0.166,Y -396.011,Z 1757.576,A 0.000,B 0.000,C 90.000,E1 283.647} C_DIS
LIN {X -0.085,Y -396.186,Z 1757.573,A 0.000,B 0.000,C 90.000,E1 283.119} C_DIS
LIN {X 0.054,Y -395.935,Z 1757.570,A 0.000,B 0.000,C 90.000,E1 282.535} C_DIS
LIN {X -0.191,Y -395.321,Z 1757.567,A 0.000,B 0.000,C 90.000,E1 282.007} C_DIS
LIN {X -0.051,Y -394.214,Z 1757.563,A 0.000,B 0.000,C 90.000,E1 281.422} C_DIS
LIN {X 0.085,Y -392.651,Z 1757.560,A 0.000,B 0.000,C 90.000,E1 280.838} C_DIS
LIN {X -0.172,Y -390.555,Z 1757.557,A 0.000,B 0.000,C 90.000,E1 280.310} C_DIS
LIN {X -0.071,Y -386.496,Z 1757.552,A 0.000,B 0.000,C 90.000,E1 279.443} C_DIS
LIN {X 0.087,Y -375.840,Z 1757.541,A 0.000,B 0.000,C 90.000,E1 277.409} C_DIS
LIN {X 0.054,Y -372.422,Z 1757.538,A 0.000,B 0.000,C 90.000,E1 276.834} C_DIS
LIN {X 0.003,Y -368.442,Z 1757.535,A 0.000,B 0.000,C 90.000,E1 276.258} C_DIS
LIN {X -0.068,Y -363.816,Z 1757.531,A 0.000,B 0.000,C 90.000,E1 275.682} C_DIS
LIN {X -0.163,Y -358.370,Z 1757.528,A 0.000,B 0.000,C 90.000,E1 275.106} C_DIS
LIN {X -0.080,Y -352.509,Z 1757.525,A 0.000,B 0.000,C 90.000,E1 274.531} C_DIS
LIN {X -0.078,Y -346.492,Z 1757.522,A 0.000,B 0.000,C 90.000,E1 274.012} C_DIS
LIN {X 0.118,Y -340.383,Z 1757.520,A 0.000,B 0.000,C 90.000,E1 273.498} C_DIS
LIN {X -0.005,Y -331.017,Z 1757.516,A 0.000,B 0.000,C 90.000,E1 272.865} C_DIS
LIN {X 0.037,Y -324.716,Z 1757.514,A 0.000,B 0.000,C 90.000,E1 272.465} C_DIS
LIN {X -0.044,Y -318.080,Z 1757.512,A 0.000,B 0.000,C 90.000,E1 272.121} C_DIS
LIN {X 0.122,Y -311.201,Z 1757.510,A 0.000,B 0.000,C 90.000,E1 271.776} C_DIS
LIN {X -0.103,Y -303.977,Z 1757.509,A 0.000,B 0.000,C 90.000,E1 271.547} C_DIS
LIN {X 0.013,Y -292.896,Z 1757.507,A 0.000,B 0.000,C 90.000,E1 271.203} C_DIS
LIN {X -0.079,Y -282.067,Z 1757.505,A 0.000,B 0.000,C 90.000,E1 270.974} C_DIS
LIN {X 0.047,Y -269.430,Z 1757.504,A 0.000,B 0.000,C 90.000,E1 270.745} C_DIS
LIN {X 0.079,Y -254.347,Z 1757.503,A 0.000,B 0.000,C 90.000,E1 270.573} C_DIS
LIN {X -0.095,Y -240.758,Z 1757.503,A 0.000,B 0.000,C 90.000,E1 270.516} C_DIS
LIN {X 0.049,Y -234.251,Z 1757.503,A 0.000,B 0.000,C 90.000,E1 270.458} C_DIS
LIN {X 0.001,Y -181.570,Z 1757.503,A 0.000,B 0.000,C 90.000,E1 270.458} C_DIS
LIN {X -0.075,Y -181.200,Z 1757.491,A 0.000,B 0.000,C 90.000,E1 268.453} C_DIS
LIN {X -0.017,Y -180.874,Z 1757.473,A 0.000,B 0.000,C 90.000,E1 265.065} C_DIS
LIN {X 0.039,Y -178.991,Z 1757.444,A 0.000,B 0.000,C 90.000,E1 259.982} C_DIS
LIN {X 0.051,Y -177.978,Z 1757.435,A 0.000,B 0.000,C 90.000,E1 258.285} C_DIS
LIN {X 0.021,Y -175.622,Z 1757.411,A 0.000,B 0.000,C 90.000,E1 254.047} C_DIS
LIN {X 0.081,Y -172.343,Z 1757.388,A 0.000,B 0.000,C 90.000,E1 249.752} C_DIS
LIN {X 0.059,Y -171.819,Z 1757.383,A 0.000,B 0.000,C 90.000,E1 248.901} C_DIS
LIN {X 0.066,Y -170.287,Z 1757.373,A 0.000,B 0.000,C 90.000,E1 247.177} C_DIS
LIN {X 0.002,Y -166.825,Z 1757.349,A 0.000,B 0.000,C 90.000,E1 242.871} C_DIS
LIN {X -0.080,Y -162.808,Z 1757.325,A 0.000,B 0.000,C 90.000,E1 238.535} C_DIS
LIN {X -0.016,Y -161.495,Z 1757.315,A 0.000,B 0.000,C 90.000,E1 236.755} C_DIS
LIN {X -0.063,Y -157.491,Z 1757.291,A 0.000,B 0.000,C 90.000,E1 232.351} C_DIS
LIN {X -0.028,Y -155.510,Z 1757.276,A 0.000,B 0.000,C 90.000,E1 229.666} C_DIS
LIN {X 0.022,Y -151.812,Z 1757.251,A 0.000,B 0.000,C 90.000,E1 225.162} C_DIS
LIN {X 0.034,Y -150.024,Z 1757.236,A 0.000,B 0.000,C 90.000,E1 222.447} C_DIS
LIN {X 0.065,Y -146.845,Z 1757.211,A 0.000,B 0.000,C 90.000,E1 217.890} C_DIS
LIN {X -0.033,Y -145.427,Z 1757.195,A 0.000,B 0.000,C 90.000,E1 215.185} C_DIS
LIN {X -0.037,Y -142.852,Z 1757.170,A 0.000,B 0.000,C 90.000,E1 210.590} C_DIS
LIN {X 0.015,Y -141.467,Z 1757.149,A 0.000,B 0.000,C 90.000,E1 206.873} C_DIS
LIN {X 0.007,Y -139.377,Z 1757.113,A 0.000,B 0.000,C 90.000,E1 200.375} C_DIS
LIN {X -0.004,Y -138.829,Z 1757.098,A 0.000,B 0.000,C 90.000,E1 197.583} C_DIS
LIN {X -0.076,Y -138.353,Z 1757.056,A 0.000,B 0.000,C 90.000,E1 190.141} C_DIS
LIN {X 0.059,Y -139.528,Z 1757.004,A 0.000,B 0.000,C 90.000,E1 180.745} C_DIS
LIN {X 0.012,Y -141.203,Z 1756.973,A 0.000,B 0.000,C 90.000,E1 175.179} C_DIS
LIN {X -0.029,Y -142.578,Z 1756.958,A 0.000,B 0.000,C 90.000,E1 172.413} C_DIS
LIN {X 0.067,Y -144.870,Z 1756.932,A 0.000,B 0.000,C 90.000,E1 167.757} C_DIS
LIN {X 0.022,Y -147.498,Z 1756.912,A 0.000,B 0.000,C 90.000,E1 164.102} C_DIS
LIN {X -0.045,Y -150.088,Z 1756.891,A 0.000,B 0.000,C 90.000,E1 160.477} C_DIS
LIN {X -0.032,Y -153.440,Z 1756.871,A 0.000,B 0.000,C 90.000,E1 156.847} C_DIS
LIN {X -0.038,Y -157.804,Z 1756.846,A 0.000,B 0.000,C 90.000,E1 152.359} C_DIS
LIN {X -0.005,Y -162.085,Z 1756.827,A 0.000,B 0.000,C 90.000,E1 148.791} C_DIS
LIN {X 0.019,Y -166.283,Z 1756.807,A 0.000,B 0.000,C 90.000,E1 145.261} C_DIS
LIN {X 0.017,Y -171.302,Z 1756.788,A 0.000,B 0.000,C 90.000,E1 141.778} C_DIS
LIN {X 0.051,Y -176.197,Z 1756.769,A 0.000,B 0.000,C 90.000,E1 138.324} C_DIS
LIN {X -0.083,Y -180.473,Z 1756.754,A 0.000,B 0.000,C 90.000,E1 135.810} C_DIS
LIN {X 0.029,Y -185.877,Z 1756.736,A 0.000,B 0.000,C 90.000,E1 132.405} C_DIS
LIN {X -0.056,Y -190.502,Z 1756.722,A 0.000,B 0.000,C 90.000,E1 129.930} C_DIS
LIN {X 0.122,Y -196.254,Z 1756.703,A 0.000,B 0.000,C 90.000,E1 126.583} C_DIS
LIN {X -0.078,Y -201.060,Z 1756.690,A 0.000,B 0.000,C 90.000,E1 124.199} C_DIS
LIN {X 0.124,Y -206.987,Z 1756.672,A 0.000,B 0.000,C 90.000,E1 120.924} C_DIS
LIN {X -0.020,Y -210.572,Z 1756.662,A 0.000,B 0.000,C 90.000,E1 119.205} C_DIS
LIN {X -0.080,Y -336.597,Z 1756.662,A 0.000,B 0.000,C 90.000,E1 119.205} C_DIS
LIN {X 0.059,Y -341.592,Z 1756.661,A 0.000,B 0.000,C 90.000,E1 119.027} C_DIS
LIN {X 0.067,Y -343.973,Z 1756.660,A 0.000,B 0.000,C 90.000,E1 118.871} C_DIS
LIN {X 0.050,Y -347.177,Z 1756.659,A 0.000,B 0.000,C 90.000,E1 118.565} C_DIS
LIN {X 0.088,Y -350.713,Z 1756.656,A 0.000,B 0.000,C 90.000,E1 118.025} C_DIS
LIN {X 0.002,Y -365.397,Z 1756.639,A 0.000,B 0.000,C 90.000,E1 115.027} C_DIS
LIN {X -0.031,Y -380.184,Z 1756.624,A 0.000,B 0.000,C 90.000,E1 112.386} C_DIS
LIN {X 0.110,Y -394.733,Z 1756.612,A 0.000,B 0.000,C 90.000,E1 110.066} C_DIS
LIN {X 0.118,Y -410.704,Z 1756.599,A 0.000,B 0.000,C 90.000,E1 107.819} C_DIS
LIN {X -0.139,Y -428.211,Z 1756.587,A 0.000,B 0.000,C 90.000,E1 105.662} C_DIS
LIN {X -0.186,Y -447.336,Z 1756.575,A 0.000,B 0.000,C 90.000,E1 103.536} C_DIS
LIN {X -0.116,Y -467.384,Z 1756.564,A 0.000,B 0.000,C 90.000,E1 101.535} C_DIS
LIN {X 0.092,Y -498.396,Z 1756.549,A 0.000,B 0.000,C 90.000,E1 98.803} C_DIS
LIN {X -0.135,Y -511.390,Z 1756.543,A 0.000,B 0.000,C 90.000,E1 97.757} C_DIS
LIN {X 0.155,Y -514.865,Z 1756.541,A 0.000,B 0.000,C 90.000,E1 97.296} C_DIS
LIN {X 0.046,Y -516.117,Z 1756.539,A 0.000,B 0.000,C 90.000,E1 97.068} C_DIS
LIN {X 0.001,Y -517.013,Z 1756.538,A 0.000,B 0.000,C 90.000,E1 96.834} C_DIS
LIN {X -0.127,Y -517.914,Z 1756.535,A 0.000,B 0.000,C 90.000,E1 96.372} C_DIS
LIN {X 0.263,Y -517.758,Z 1756.533,A 0.000,B 0.000,C 90.000,E1 95.853} C_DIS
LIN {X 0.143,Y -516.522,Z 1756.530,A 0.000,B 0.000,C 90.000,E1 95.391} C_DIS
LIN {X 0.059,Y -515.434,Z 1756.529,A 0.000,B 0.000,C 90.000,E1 95.163} C_DIS
LIN {X -0.068,Y -512.275,Z 1756.526,A 0.000,B 0.000,C 90.000,E1 94.702} C_DIS
LIN {X 0.184,Y -498.887,Z 1756.515,A 0.000,B 0.000,C 90.000,E1 92.751} C_DIS
LIN {X 0.059,Y -490.205,Z 1756.509,A 0.000,B 0.000,C 90.000,E1 91.547} C_DIS
LIN {X -0.044,Y -477.630,Z 1756.499,A 0.000,B 0.000,C 90.000,E1 89.828} C_DIS
LIN {X -0.187,Y -466.668,Z 1756.491,A 0.000,B 0.000,C 90.000,E1 88.339} C_DIS
LIN {X 0.210,Y -453.807,Z 1756.481,A 0.000,B 0.000,C 90.000,E1 86.502} C_DIS
LIN {X -0.107,Y -441.009,Z 1756.471,A 0.000,B 0.000,C 90.000,E1 84.723} C_DIS
LIN {X -0.023,Y -426.554,Z 1756.459,A 0.000,B 0.000,C 90.000,E1 82.591} C_DIS
LIN {X 0.148,Y -407.474,Z 1756.442,A 0.000,B 0.000,C 90.000,E1 79.577} C_DIS
LIN {X -0.132,Y -391.040,Z 1756.427,A 0.000,B 0.000,C 90.000,E1 76.825} C_DIS
LIN {X 0.133,Y -377.003,Z 1756.412,A 0.000,B 0.000,C 90.000,E1 74.212} C_DIS
LIN {X 0.039,Y -364.983,Z 1756.399,A 0.000,B 0.000,C 90.000,E1 71.891} C_DIS
LIN {X -0.005,Y -353.323,Z 1756.386,A 0.000,B 0.000,C 90.000,E1 69.518} C_DIS
LIN {X -0.049,Y -339.294,Z 1756.369,A 0.000,B 0.000,C 90.000,E1 66.485} C_DIS
LIN {X 0.155,Y -329.807,Z 1756.357,A 0.000,B 0.000,C 90.000,E1 64.280} C_DIS
LIN {X 0.083,Y -319.121,Z 1756.343,A 0.000,B 0.000,C 90.000,E1 61.769} C_DIS
LIN {X -0.124,Y -312.308,Z 1756.334,A 0.000,B 0.000,C 90.000,E1 60.205} C_DIS
LIN {X 0.147,Y -305.201,Z 1756.325,A 0.000,B 0.000,C 90.000,E1 58.535} C_DIS
LIN {X -0.183,Y -294.917,Z 1756.313,A 0.000,B 0.000,C 90.000,E1 56.294} C_DIS
LIN {X -0.019,Y -283.388,Z 1756.298,A 0.000,B 0.000,C 90.000,E1 53.577} C_DIS
LIN {X 0.010,Y -270.714,Z 1756.281,A 0.000,B 0.000,C 90.000,E1 50.481} C_DIS
LIN {X -0.011,Y -259.995,Z 1756.265,A 0.000,B 0.000,C 90.000,E1 47.676} C_DIS
LIN {X 0.009,Y -252.130,Z 1756.253,A 0.000,B 0.000,C 90.000,E1 45.526} C_DIS
LIN {X 0.021,Y -240.764,Z 1756.235,A 0.000,B 0.000,C 90.000,E1 42.243} C_DIS
LIN {X -0.069,Y -229.959,Z 1756.216,A 0.000,B 0.000,C 90.000,E1 38.910} C_DIS
LIN {X -0.007,Y -220.954,Z 1756.199,A 0.000,B 0.000,C 90.000,E1 35.851} C_DIS
LIN {X 0.007,Y -212.614,Z 1756.182,A 0.000,B 0.000,C 90.000,E1 32.752} C_DIS
LIN {X -0.042,Y -205.126,Z 1756.164,A 0.000,B 0.000,C 90.000,E1 29.617} C_DIS
LIN {X -0.021,Y -198.274,Z 1756.147,A 0.000,B 0.000,C 90.000,E1 26.411} C_DIS
LIN {X 0.013,Y -192.181,Z 1756.129,A 0.000,B 0.000,C 90.000,E1 23.153} C_DIS
LIN {X -0.063,Y -186.895,Z 1756.110,A 0.000,B 0.000,C 90.000,E1 19.885} C_DIS
LIN {X -0.050,Y -182.396,Z 1756.092,A 0.000,B 0.000,C 90.000,E1 16.551} C_DIS
LIN {X -0.011,Y -178.843,Z 1756.073,A 0.000,B 0.000,C 90.000,E1 13.175} C_DIS
LIN {X 0.042,Y -175.414,Z 1756.050,A 0.000,B 0.000,C 90.000,E1 8.916} C_DIS
LIN {X 0.044,Y -172.615,Z 1756.021,A 0.000,B 0.000,C 90.000,E1 3.784} C_DIS
LIN {X -0.048,Y -171.293,Z 1755.983,A 0.000,B 0.000,C 90.000,E1 356.963} C_DIS
LIN {X -0.041,Y -172.122,Z 1755.935,A 0.000,B 0.000,C 90.000,E1 348.342} C_DIS
LIN {X 0.016,Y -174.347,Z 1755.902,A 0.000,B 0.000,C 90.000,E1 342.308} C_DIS
LIN {X 0.030,Y -177.753,Z 1755.873,A 0.000,B 0.000,C 90.000,E1 337.177} C_DIS
LIN {X 0.000,Y -181.413,Z 1755.850,A 0.000,B 0.000,C 90.000,E1 332.948} C_DIS
LIN {X 0.018,Y -186.135,Z 1755.826,A 0.000,B 0.000,C 90.000,E1 328.742} C_DIS
LIN {X 0.105,Y -190.866,Z 1755.808,A 0.000,B 0.000,C 90.000,E1 325.388} C_DIS
LIN {X 0.064,Y -196.539,Z 1755.790,A 0.000,B 0.000,C 90.000,E1 322.110} C_DIS
LIN {X -0.055,Y -201.488,Z 1755.776,A 0.000,B 0.000,C 90.000,E1 319.703} C_DIS
LIN {X 0.059,Y -209.246,Z 1755.758,A 0.000,B 0.000,C 90.000,E1 316.458} C_DIS
LIN {X -0.056,Y -214.762,Z 1755.747,A 0.000,B 0.000,C 90.000,E1 314.514} C_DIS
LIN {X 0.069,Y -221.002,Z 1755.736,A 0.000,B 0.000,C 90.000,E1 312.528} C_DIS
LIN {X 0.000,Y -228.114,Z 1755.726,A 0.000,B 0.000,C 90.000,E1 310.620} C_DIS
LIN {X -0.069,Y -234.609,Z 1755.717,A 0.000,B 0.000,C 90.000,E1 309.116} C_DIS
LIN {X -0.043,Y -243.765,Z 1755.707,A 0.000,B 0.000,C 90.000,E1 307.237} C_DIS
LIN {X -0.120,Y -258.104,Z 1755.693,A 0.000,B 0.000,C 90.000,E1 304.692} C_DIS
LIN {X 0.130,Y -276.332,Z 1755.677,A 0.000,B 0.000,C 90.000,E1 301.799} C_DIS
LIN {X 0.045,Y -296.079,Z 1755.662,A 0.000,B 0.000,C 90.000,E1 299.077} C_DIS
LIN {X 0.131,Y -314.101,Z 1755.649,A 0.000,B 0.000,C 90.000,E1 296.744} C_DIS
LIN {X -0.014,Y -330.023,Z 1755.638,A 0.000,B 0.000,C 90.000,E1 294.847} C_DIS
LIN {X 0.159,Y -343.093,Z 1755.629,A 0.000,B 0.000,C 90.000,E1 293.259} C_DIS
LIN {X -0.103,Y -355.958,Z 1755.621,A 0.000,B 0.000,C 90.000,E1 291.770} C_DIS
LIN {X -0.033,Y -365.737,Z 1755.614,A 0.000,B 0.000,C 90.000,E1 290.556} C_DIS
LIN {X 0.206,Y -372.525,Z 1755.609,A 0.000,B 0.000,C 90.000,E1 289.631} C_DIS
LIN {X 0.023,Y -378.628,Z 1755.604,A 0.000,B 0.000,C 90.000,E1 288.779} C_DIS
LIN {X 0.134,Y -382.212,Z 1755.601,A 0.000,B 0.000,C 90.000,E1 288.181} C_DIS
LIN {X -0.096,Y -385.351,Z 1755.598,A 0.000,B 0.000,C 90.000,E1 287.638} C_DIS
LIN {X 0.208,Y -389.232,Z 1755.593,A 0.000,B 0.000,C 90.000,E1 286.732} C_DIS
LIN {X 0.058,Y -392.228,Z 1755.588,A 0.000,B 0.000,C 90.000,E1 285.898} C_DIS
LIN {X -0.227,Y -393.779,Z 1755.585,A 0.000,B 0.000,C 90.000,E1 285.371} C_DIS
LIN {X -0.016,Y -394.988,Z 1755.582,A 0.000,B 0.000,C 90.000,E1 284.773} C_DIS
LIN {X 0.106,Y -395.860,Z 1755.579,A 0.000,B 0.000,C 90.000,E1 284.189} C_DIS
LIN {X -0.052,Y -396.357,Z 1755.576,A 0.000,B 0.000,C 90.000,E1 283.647} C_DIS
LIN {X 0.084,Y -396.509,Z 1755.573,A 0.000,B 0.000,C 90.000,E1 283.063} C_DIS
LIN {X -0.160,Y -396.218,Z 1755.569,A 0.000,B 0.000,C 90.000,E1 282.535} C_DIS
LIN {X -0.016,Y -395.557,Z 1755.566,A 0.000,B 0.000,C 90.000,E1 281.951} C_DIS
LIN {X 0.126,Y -394.405,Z 1755.563,A 0.000,B 0.000,C 90.000,E1 281.366} C_DIS
LIN {X -0.123,Y -392.745,Z 1755.560,A 0.000,B 0.000,C 90.000,E1 280.838} C_DIS
LIN {X 0.008,Y -390.581,Z 1755.557,A 0.000,B 0.000,C 90.000,E1 280.254} C_DIS
LIN {X 0.125,Y -387.904,Z 1755.554,A 0.000,B 0.000,C 90.000,E1 279.670} C_DIS
LIN {X -0.111,Y -375.731,Z 1755.541,A 0.000,B 0.000,C 90.000,E1 277.409} C_DIS
LIN {X -0.144,Y -372.310,Z 1755.538,A 0.000,B 0.000,C 90.000,E1 276.834} C_DIS
LIN {X 0.172,Y -368.284,Z 1755.535,A 0.000,B 0.000,C 90.000,E1 276.201} C_DIS
LIN {X 0.099,Y -363.539,Z 1755.531,A 0.000,B 0.000,C 90.000,E1 275.625} C_DIS
LIN {X 0.001,Y -358.092,Z 1755.528,A 0.000,B 0.000,C 90.000,E1 275.049} C_DIS
LIN {X 0.086,Y -352.138,Z 1755.525,A 0.000,B 0.000,C 90.000,E1 274.473} C_DIS
LIN {X 0.108,Y -346.144,Z 1755.522,A 0.000,B 0.000,C 90.000,E1 273.955} C_DIS
LIN {X -0.038,Y -339.964,Z 1755.519,A 0.000,B 0.000,C 90.000,E1 273.498} C_DIS
LIN {X -0.123,Y -330.644,Z 1755.516,A 0.000,B 0.000,C 90.000,E1 272.865} C_DIS
LIN {X -0.061,Y -324.210,Z 1755.514,A 0.000,B 0.000,C 90.000,E1 272.465} C_DIS
LIN {X -0.130,Y -317.519,Z 1755.512,A 0.000,B 0.000,C 90.000,E1 272.121} C_DIS
LIN {X 0.029,Y -310.482,Z 1755.510,A 0.000,B 0.000,C 90.000,E1 271.776} C_DIS
LIN {X 0.127,Y -303.221,Z 1755.508,A 0.000,B 0.000,C 90.000,E1 271.489} C_DIS
LIN {X -0.019,Y -292.067,Z 1755.507,A 0.000,B 0.000,C 90.000,E1 271.203} C_DIS
LIN {X -0.078,Y -281.415,Z 1755.505,A 0.000,B 0.000,C 90.000,E1 270.974} C_DIS
LIN {X 0.097,Y -273.383,Z 1755.505,A 0.000,B 0.000,C 90.000,E1 270.802} C_DIS
LIN {X 0.097,Y -258.812,Z 1755.504,A 0.000,B 0.000,C 90.000,E1 270.630} C_DIS
LIN {X -0.042,Y -240.055,Z 1755.503,A 0.000,B 0.000,C 90.000,E1 270.516} C_DIS
LIN {X -0.089,Y -237.340,Z 1755.503,A 0.000,B 0.000,C 90.000,E1 270.516} C_DIS
LIN {X 0.078,Y -181.567,Z 1755.503,A 0.000,B 0.000,C 90.000,E1 270.458} C_DIS
LIN {X -0.005,Y -181.114,Z 1755.489,A 0.000,B 0.000,C 90.000,E1 267.936} C_DIS
LIN {X -0.017,Y -180.906,Z 1755.474,A 0.000,B 0.000,C 90.000,E1 265.412} C_DIS
